LIN {X 0,Y 524.24,Z 195.314,A -85,B 0,C 180,E1 -4882.904,E2 -4882.904} C_VEL
LIN {X 0,Y 525.954,Z 203.789,A -85,B 0,C 180,E1 -4883.085,E2 -4883.085} C_VEL
LIN {X 0,Y 525.499,Z 302.73,A -85,B 0,C 180,E1 -4884.494,E2 -4884.494} C_VEL
LIN {X 0,Y 525.358,Z 316.211,A -85,B 0,C 180,E1 -4884.854,E2 -4884.854} C_VEL
LIN {X 0,Y 525.146,Z 328.864,A -85,B 0,C 180,E1 -4885.357,E2 -4885.357} C_VEL
LIN {X 0,Y 524.878,Z 340.909,A -85,B 0,C 180,E1 -4886.009,E2 -4886.009} C_VEL
LIN {X 0,Y 524.614,Z 351.923,A -85,B 0,C 180,E1 -4886.773,E2 -4886.773} C_VEL
LIN {X 0,Y 524.367,Z 361.654,A -85,B 0,C 180,E1 -4887.611,E2 -4887.611} C_VEL
LIN {X 0,Y 524.142,Z 371.309,A -85,B 0,C 180,E1 -4888.643,E2 -4888.643} C_VEL
LIN {X 0,Y 523.923,Z 379.749,A -85,B 0,C 180,E1 -4889.757,E2 -4889.757} C_VEL
LIN {X 0,Y 523.73,Z 386.278,A -85,B 0,C 180,E1 -4890.815,E2 -4890.815} C_VEL
LIN {X 0,Y 523.699,Z 387.83,A -85,B 0,C 180,E1 -4891.105,E2 -4891.105} C_VEL
LIN {X 0,Y 522.987,Z 390.737,A -85,B 0,C 180,E1 -4891.663,E2 -4891.663} C_VEL
LIN {X 0,Y 520.036,Z 395.032,A -85,B 0,C 180,E1 -4892.59,E2 -4892.59} C_VEL
LIN {X 0,Y 517.078,Z 398.654,A -85,B 0,C 180,E1 -4893.561,E2 -4893.561} C_VEL
LIN {X 0,Y 516.367,Z 400.435,A -85,B 0,C 180,E1 -4894.182,E2 -4894.182} C_VEL
LIN {X 0,Y 516.321,Z 402.767,A -85,B 0,C 180,E1 -4895.244,E2 -4895.244} C_VEL
LIN {X 0,Y 516.258,Z 404.817,A -85,B 0,C 180,E1 -4896.797,E2 -4896.797} C_VEL
LIN {X 0,Y 516.242,Z 405.275,A -85,B 0,C 180,E1 -4897.852,E2 -4897.852} C_VEL
LIN {X 0,Y 516.25,Z 404.907,A -85,B 0,C 180,E1 -4899.107,E2 -4899.107} C_VEL
LIN {X 0,Y 516.299,Z 403.557,A -85,B 0,C 180,E1 -4900.334,E2 -4900.334} C_VEL
LIN {X 0,Y 516.377,Z 400.571,A -85,B 0,C 180,E1 -4901.828,E2 -4901.828} C_VEL
LIN {X 0,Y 516.471,Z 397.517,A -85,B 0,C 180,E1 -4902.874,E2 -4902.874} C_VEL
LIN {X 0,Y 516.547,Z 392.428,A -85,B 0,C 180,E1 -4904.2,E2 -4904.2} C_VEL
LIN {X 0,Y 516.706,Z 385.586,A -85,B 0,C 180,E1 -4905.556,E2 -4905.556} C_VEL
LIN {X 0,Y 516.897,Z 378.682,A -85,B 0,C 180,E1 -4906.647,E2 -4906.647} C_VEL
LIN {X 0,Y 517.166,Z 370.161,A -85,B 0,C 180,E1 -4907.745,E2 -4907.745} C_VEL
LIN {X 0,Y 517.452,Z 359.972,A -85,B 0,C 180,E1 -4908.798,E2 -4908.798} C_VEL
LIN {X 0,Y 517.679,Z 349.531,A -85,B 0,C 180,E1 -4909.669,E2 -4909.669} C_VEL
LIN {X 0,Y 517.992,Z 338.867,A -85,B 0,C 180,E1 -4910.381,E2 -4910.381} C_VEL
LIN {X 0,Y 518.301,Z 327.456,A -85,B 0,C 180,E1 -4910.974,E2 -4910.974} C_VEL
LIN {X 0,Y 518.454,Z 313.875,A -85,B 0,C 180,E1 -4911.494,E2 -4911.494} C_VEL
LIN {X 0,Y 518.631,Z 301.35,A -85,B 0,C 180,E1 -4911.81,E2 -4911.81} C_VEL
LIN {X 0,Y 519.072,Z 204.764,A -85,B 0,C 180,E1 -4913.193,E2 -4913.193} C_VEL
LIN {X 0,Y 517.223,Z 195.581,A -85,B 0,C 180,E1 -4913.39,E2 -4913.39} C_VEL
LIN {X 0,Y 516.967,Z 190.248,A -85,B 0,C 180,E1 -4914.482,E2 -4914.482} C_VEL
LIN {X 0,Y 516.894,Z 190.102,A -85,B 0,C 180,E1 -4917.457,E2 -4917.457} C_VEL
LIN {X 0,Y 516.921,Z 190.092,A -85,B 0,C 180,E1 -4920.696,E2 -4920.696} C_VEL
LIN {X 0,Y 516.897,Z 190.094,A -85,B 0,C 180,E1 -4923.815,E2 -4923.815} C_VEL
LIN {X 0,Y 516.858,Z 190.103,A -85,B 0,C 180,E1 -4926.776,E2 -4926.776} C_VEL
LIN {X 0,Y 516.938,Z 190.088,A -85,B 0,C 180,E1 -4929.733,E2 -4929.733} C_VEL
LIN {X 0,Y 516.896,Z 190.097,A -85,B 0,C 180,E1 -4932.595,E2 -4932.595} C_VEL
LIN {X 0,Y 516.941,Z 190.094,A -85,B 0,C 180,E1 -4935.03,E2 -4935.03} C_VEL
LIN {X 0,Y 516.968,Z 190.086,A -85,B 0,C 180,E1 -4938.234,E2 -4938.234} C_VEL
LIN {X 0,Y 516.956,Z 190.086,A -85,B 0,C 180,E1 -4941.4,E2 -4941.4} C_VEL
LIN {X 0,Y 517.025,Z 190.085,A -85,B 0,C 180,E1 -4944.54,E2 -4944.54} C_VEL
LIN {X 0,Y 517.082,Z 190.07,A -85,B 0,C 180,E1 -4947.663,E2 -4947.663} C_VEL
LIN {X 0,Y 517.092,Z 190.073,A -85,B 0,C 180,E1 -4950.779,E2 -4950.779} C_VEL
LIN {X 0,Y 516.975,Z 190.084,A -85,B 0,C 180,E1 -4953.117,E2 -4953.117} C_VEL
LIN {X 0,Y 516.991,Z 190.089,A -85,B 0,C 180,E1 -4956.244,E2 -4956.244} C_VEL
LIN {X 0,Y 516.943,Z 190.087,A -85,B 0,C 180,E1 -4959.39,E2 -4959.39} C_VEL
LIN {X 0,Y 516.954,Z 190.089,A -85,B 0,C 180,E1 -4961.807,E2 -4961.807} C_VEL
LIN {X 0,Y 516.941,Z 190.087,A -85,B 0,C 180,E1 -4965.144,E2 -4965.144} C_VEL
LIN {X 0,Y 516.914,Z 190.098,A -85,B 0,C 180,E1 -4968.223,E2 -4968.223} C_VEL
LIN {X 0,Y 516.907,Z 190.093,A -85,B 0,C 180,E1 -4970.702,E2 -4970.702} C_VEL
LIN {X 0,Y 516.887,Z 190.101,A -85,B 0,C 180,E1 -4974.073,E2 -4974.073} C_VEL
LIN {X 0,Y 516.89,Z 190.094,A -85,B 0,C 180,E1 -4976.66,E2 -4976.66} C_VEL
LIN {X 0,Y 516.909,Z 190.096,A -85,B 0,C 180,E1 -4979.523,E2 -4979.523} C_VEL
LIN {X 0,Y 516.898,Z 190.093,A -85,B 0,C 180,E1 -4982.543,E2 -4982.543} C_VEL
LIN {X 0,Y 516.866,Z 190.101,A -85,B 0,C 180,E1 -4985.329,E2 -4985.329} C_VEL
LIN {X 0,Y 516.88,Z 190.099,A -85,B 0,C 180,E1 -4987.943,E2 -4987.943} C_VEL
LIN {X 0,Y 516.866,Z 190.097,A -85,B 0,C 180,E1 -4990.744,E2 -4990.744} C_VEL
LIN {X 0,Y 516.861,Z 190.099,A -85,B 0,C 180,E1 -4992.834,E2 -4992.834} C_VEL
LIN {X 0,Y 516.898,Z 190.096,A -85,B 0,C 180,E1 -4995.007,E2 -4995.007} C_VEL
LIN {X 0,Y 516.904,Z 190.092,A -85,B 0,C 180,E1 -4998.4,E2 -4998.4} C_VEL
LIN {X 0,Y 516.879,Z 190.105,A -85,B 0,C 180,E1 -5001.284,E2 -5001.284} C_VEL
LIN {X 0,Y 516.87,Z 190.096,A -85,B 0,C 180,E1 -5004.22,E2 -5004.22} C_VEL
LIN {X 0,Y 516.883,Z 190.102,A -85,B 0,C 180,E1 -5007.052,E2 -5007.052} C_VEL
LIN {X 0,Y 516.869,Z 190.097,A -85,B 0,C 180,E1 -5009.795,E2 -5009.795} C_VEL
LIN {X 0,Y 516.885,Z 190.096,A -85,B 0,C 180,E1 -5012.465,E2 -5012.465} C_VEL
LIN {X 0,Y 516.853,Z 190.106,A -85,B 0,C 180,E1 -5015.069,E2 -5015.069} C_VEL
LIN {X 0,Y 516.872,Z 190.097,A -85,B 0,C 180,E1 -5017.622,E2 -5017.622} C_VEL
LIN {X 0,Y 516.932,Z 190.089,A -85,B 0,C 180,E1 -5020.13,E2 -5020.13} C_VEL
LIN {X 0,Y 516.896,Z 190.099,A -85,B 0,C 180,E1 -5022.595,E2 -5022.595} C_VEL
LIN {X 0,Y 516.935,Z 190.093,A -85,B 0,C 180,E1 -5025.03,E2 -5025.03} C_VEL
LIN {X 0,Y 516.97,Z 190.087,A -85,B 0,C 180,E1 -5028.234,E2 -5028.234} C_VEL
LIN {X 0,Y 516.956,Z 190.086,A -85,B 0,C 180,E1 -5031.399,E2 -5031.399} C_VEL
LIN {X 0,Y 517.014,Z 190.087,A -85,B 0,C 180,E1 -5034.54,E2 -5034.54} C_VEL
LIN {X 0,Y 517.082,Z 190.07,A -85,B 0,C 180,E1 -5037.663,E2 -5037.663} C_VEL
LIN {X 0,Y 517.069,Z 190.075,A -85,B 0,C 180,E1 -5040.779,E2 -5040.779} C_VEL
LIN {X 0,Y 516.949,Z 190.087,A -85,B 0,C 180,E1 -5043.117,E2 -5043.117} C_VEL
LIN {X 0,Y 516.975,Z 190.092,A -85,B 0,C 180,E1 -5046.244,E2 -5046.244} C_VEL
LIN {X 0,Y 516.939,Z 190.088,A -85,B 0,C 180,E1 -5049.39,E2 -5049.39} C_VEL
LIN {X 0,Y 516.956,Z 190.091,A -85,B 0,C 180,E1 -5051.807,E2 -5051.807} C_VEL
LIN {X 0,Y 516.943,Z 190.087,A -85,B 0,C 180,E1 -5055.144,E2 -5055.144} C_VEL
LIN {X 0,Y 516.879,Z 190.1,A -85,B 0,C 180,E1 -5058.224,E2 -5058.224} C_VEL
LIN {X 0,Y 516.903,Z 190.093,A -85,B 0,C 180,E1 -5060.702,E2 -5060.702} C_VEL
LIN {X 0,Y 516.859,Z 190.099,A -85,B 0,C 180,E1 -5063.224,E2 -5063.224} C_VEL
LIN {X 0,Y 516.884,Z 190.097,A -85,B 0,C 180,E1 -5066.182,E2 -5066.182} C_VEL
LIN {X 0,Y 516.906,Z 190.096,A -85,B 0,C 180,E1 -5069.306,E2 -5069.306} C_VEL
LIN {X 0,Y 516.896,Z 190.093,A -85,B 0,C 180,E1 -5072.543,E2 -5072.543} C_VEL
LIN {X 0,Y 516.863,Z 190.103,A -85,B 0,C 180,E1 -5075.328,E2 -5075.328} C_VEL
LIN {X 0,Y 516.88,Z 190.098,A -85,B 0,C 180,E1 -5077.942,E2 -5077.942} C_VEL
LIN {X 0,Y 516.855,Z 190.099,A -85,B 0,C 180,E1 -5080.745,E2 -5080.745} C_VEL
LIN {X 0,Y 516.883,Z 190.096,A -85,B 0,C 180,E1 -5083.903,E2 -5083.903} C_VEL
LIN {X 0,Y 516.882,Z 190.095,A -85,B 0,C 180,E1 -5086.107,E2 -5086.107} C_VEL
LIN {X 0,Y 516.855,Z 190.106,A -85,B 0,C 180,E1 -5089.255,E2 -5089.255} C_VEL
LIN {X 0,Y 516.862,Z 190.098,A -85,B 0,C 180,E1 -5092.274,E2 -5092.274} C_VEL
LIN {X 0,Y 516.875,Z 190.104,A -85,B 0,C 180,E1 -5095.174,E2 -5095.174} C_VEL
LIN {X 0,Y 516.87,Z 190.098,A -85,B 0,C 180,E1 -5097.974,E2 -5097.974} C_VEL
LIN {X 0,Y 516.905,Z 190.099,A -85,B 0,C 180,E1 -5100.694,E2 -5100.694} C_VEL
LIN {X 0,Y 516.901,Z 190.178,A -85,B 0,C 180,E1 -5103.633,E2 -5103.633} C_VEL
LIN {X 0,Y 518.785,Z 200.2,A -85,B 0,C 180,E1 -5105.183,E2 -5105.183} C_VEL
LIN {X 0,Y 518.36,Z 217.704,A -85,B 0,C 180,E1 -5107.689,E2 -5107.689} C_VEL
LIN {X 0,Y 517.906,Z 238.22,A -85,B 0,C 180,E1 -5110.581,E2 -5110.581} C_VEL
LIN {X 0,Y 517.415,Z 260.123,A -85,B 0,C 180,E1 -5113.629,E2 -5113.629} C_VEL
LIN {X 0,Y 517.252,Z 267.307,A -85,B 0,C 180,E1 -5114.623,E2 -5114.623} C_VEL
LIN {X 0,Y 519.019,Z 280.709,A -85,B 0,C 180,E1 -5114.873,E2 -5114.873} C_VEL
LIN {X 0,Y 518.492,Z 377.185,A -85,B 0,C 180,E1 -5116.253,E2 -5116.253} C_VEL
LIN {X 0,Y 518.229,Z 390.964,A -85,B 0,C 180,E1 -5116.621,E2 -5116.621} C_VEL
LIN {X 0,Y 517.971,Z 403.375,A -85,B 0,C 180,E1 -5117.113,E2 -5117.113} C_VEL
LIN {X 0,Y 517.622,Z 415.512,A -85,B 0,C 180,E1 -5117.766,E2 -5117.766} C_VEL
LIN {X 0,Y 517.352,Z 426.757,A -85,B 0,C 180,E1 -5118.54,E2 -5118.54} C_VEL
LIN {X 0,Y 517.081,Z 437.113,A -85,B 0,C 180,E1 -5119.427,E2 -5119.427} C_VEL
LIN {X 0,Y 516.812,Z 446.415,A -85,B 0,C 180,E1 -5120.41,E2 -5120.41} C_VEL
LIN {X 0,Y 516.628,Z 455.472,A -85,B 0,C 180,E1 -5121.591,E2 -5121.591} C_VEL
LIN {X 0,Y 516.503,Z 462.768,A -85,B 0,C 180,E1 -5122.769,E2 -5122.769} C_VEL
LIN {X 0,Y 516.381,Z 467.688,A -85,B 0,C 180,E1 -5123.749,E2 -5123.749} C_VEL
LIN {X 0,Y 516.312,Z 472.473,A -85,B 0,C 180,E1 -5124.924,E2 -5124.924} C_VEL
LIN {X 0,Y 516.372,Z 476.135,A -85,B 0,C 180,E1 -5126.098,E2 -5126.098} C_VEL
LIN {X 0,Y 516.346,Z 478.019,A -85,B 0,C 180,E1 -5126.879,E2 -5126.879} C_VEL
LIN {X 0,Y 516.264,Z 479.427,A -85,B 0,C 180,E1 -5127.659,E2 -5127.659} C_VEL
LIN {X 0,Y 516.199,Z 481.039,A -85,B 0,C 180,E1 -5129.22,E2 -5129.22} C_VEL
LIN {X 0,Y 516.203,Z 481.252,A -85,B 0,C 180,E1 -5130,E2 -5130} C_VEL
LIN {X 0,Y 516.2,Z 481.027,A -85,B 0,C 180,E1 -5130.78,E2 -5130.78} C_VEL
LIN {X 0,Y 516.264,Z 479.391,A -85,B 0,C 180,E1 -5132.34,E2 -5132.34} C_VEL
LIN {X 0,Y 516.362,Z 477.97,A -85,B 0,C 180,E1 -5133.121,E2 -5133.121} C_VEL
LIN {X 0,Y 516.344,Z 474.975,A -85,B 0,C 180,E1 -5134.293,E2 -5134.293} C_VEL
LIN {X 0,Y 516.389,Z 470.928,A -85,B 0,C 180,E1 -5135.467,E2 -5135.467} C_VEL
LIN {X 0,Y 516.418,Z 465.656,A -85,B 0,C 180,E1 -5136.655,E2 -5136.655} C_VEL
LIN {X 0,Y 516.538,Z 459.159,A -85,B 0,C 180,E1 -5137.82,E2 -5137.82} C_VEL
LIN {X 0,Y 516.713,Z 450.992,A -85,B 0,C 180,E1 -5138.999,E2 -5138.999} C_VEL
LIN {X 0,Y 516.903,Z 442.664,A -85,B 0,C 180,E1 -5139.983,E2 -5139.983} C_VEL
LIN {X 0,Y 517.199,Z 432.511,A -85,B 0,C 180,E1 -5140.967,E2 -5140.967} C_VEL
LIN {X 0,Y 517.446,Z 421.234,A -85,B 0,C 180,E1 -5141.84,E2 -5141.84} C_VEL
LIN {X 0,Y 517.789,Z 409.771,A -85,B 0,C 180,E1 -5142.543,E2 -5142.543} C_VEL
LIN {X 0,Y 518.077,Z 397.232,A -85,B 0,C 180,E1 -5143.133,E2 -5143.133} C_VEL
LIN {X 0,Y 518.353,Z 383.87,A -85,B 0,C 180,E1 -5143.575,E2 -5143.575} C_VEL
LIN {X 0,Y 518.583,Z 370.916,A -85,B 0,C 180,E1 -5143.844,E2 -5143.844} C_VEL
LIN {X 0,Y 518.922,Z 279.596,A -85,B 0,C 180,E1 -5145.138,E2 -5145.138} C_VEL
LIN {X 0,Y 517.22,Z 266.453,A -85,B 0,C 180,E1 -5145.397,E2 -5145.397} C_VEL
LIN {X 0,Y 517.663,Z 242.885,A -85,B 0,C 180,E1 -5148.605,E2 -5148.605} C_VEL
LIN {X 0,Y 517.991,Z 221.824,A -85,B 0,C 180,E1 -5151.489,E2 -5151.489} C_VEL
LIN {X 0,Y 518.421,Z 200.841,A -85,B 0,C 180,E1 -5154.386,E2 -5154.386} C_VEL
LIN {X 0,Y 518.054,Z 195.968,A -85,B 0,C 180,E1 -5155.084,E2 -5155.084} C_VEL
LIN {X 0,Y 516.884,Z 190.1,A -85,B 0,C 180,E1 -5155.985,E2 -5155.985} C_VEL
LIN {X 0,Y 516.849,Z 190.104,A -85,B 0,C 180,E1 -5158.419,E2 -5158.419} C_VEL
LIN {X 0,Y 516.88,Z 190.104,A -85,B 0,C 180,E1 -5161.11,E2 -5161.11} C_VEL
LIN {X 0,Y 516.886,Z 190.096,A -85,B 0,C 180,E1 -5163.962,E2 -5163.962} C_VEL
LIN {X 0,Y 516.854,Z 190.107,A -85,B 0,C 180,E1 -5166.748,E2 -5166.748} C_VEL
LIN {X 0,Y 516.858,Z 190.099,A -85,B 0,C 180,E1 -5169.723,E2 -5169.723} C_VEL
LIN {X 0,Y 516.901,Z 190.093,A -85,B 0,C 180,E1 -5171.776,E2 -5171.776} C_VEL
LIN {X 0,Y 516.896,Z 190.097,A -85,B 0,C 180,E1 -5175.007,E2 -5175.007} C_VEL
LIN {X 0,Y 516.903,Z 190.099,A -85,B 0,C 180,E1 -5178.4,E2 -5178.4} C_VEL
LIN {X 0,Y 516.877,Z 190.097,A -85,B 0,C 180,E1 -5181.284,E2 -5181.284} C_VEL
LIN {X 0,Y 516.868,Z 190.105,A -85,B 0,C 180,E1 -5184.219,E2 -5184.219} C_VEL
LIN {X 0,Y 516.895,Z 190.094,A -85,B 0,C 180,E1 -5187.053,E2 -5187.053} C_VEL
LIN {X 0,Y 516.885,Z 190.099,A -85,B 0,C 180,E1 -5189.796,E2 -5189.796} C_VEL
LIN {X 0,Y 516.899,Z 190.096,A -85,B 0,C 180,E1 -5192.466,E2 -5192.466} C_VEL
LIN {X 0,Y 516.851,Z 190.1,A -85,B 0,C 180,E1 -5195.069,E2 -5195.069} C_VEL
LIN {X 0,Y 516.869,Z 190.1,A -85,B 0,C 180,E1 -5197.621,E2 -5197.621} C_VEL
LIN {X 0,Y 516.929,Z 190.096,A -85,B 0,C 180,E1 -5200.13,E2 -5200.13} C_VEL
LIN {X 0,Y 516.894,Z 190.093,A -85,B 0,C 180,E1 -5202.595,E2 -5202.595} C_VEL
LIN {X 0,Y 516.936,Z 190.089,A -85,B 0,C 180,E1 -5205.03,E2 -5205.03} C_VEL
LIN {X 0,Y 516.966,Z 190.086,A -85,B 0,C 180,E1 -5208.234,E2 -5208.234} C_VEL
LIN {X 0,Y 516.965,Z 190.09,A -85,B 0,C 180,E1 -5211.4,E2 -5211.4} C_VEL
LIN {X 0,Y 517.003,Z 190.086,A -85,B 0,C 180,E1 -5213.757,E2 -5213.757} C_VEL
LIN {X 0,Y 517.009,Z 190.081,A -85,B 0,C 180,E1 -5216.883,E2 -5216.883} C_VEL
LIN {X 0,Y 517.093,Z 190.075,A -85,B 0,C 180,E1 -5219.221,E2 -5219.221} C_VEL
LIN {X 0,Y 517.084,Z 190.071,A -85,B 0,C 180,E1 -5222.337,E2 -5222.337} C_VEL
LIN {X 0,Y 517.027,Z 190.083,A -85,B 0,C 180,E1 -5225.46,E2 -5225.46} C_VEL
LIN {X 0,Y 516.956,Z 190.089,A -85,B 0,C 180,E1 -5228.6,E2 -5228.6} C_VEL
LIN {X 0,Y 516.952,Z 190.09,A -85,B 0,C 180,E1 -5231.807,E2 -5231.807} C_VEL
LIN {X 0,Y 516.945,Z 190.096,A -85,B 0,C 180,E1 -5235.146,E2 -5235.146} C_VEL
LIN {X 0,Y 516.916,Z 190.095,A -85,B 0,C 180,E1 -5238.223,E2 -5238.223} C_VEL
LIN {X 0,Y 516.919,Z 190.099,A -85,B 0,C 180,E1 -5240.701,E2 -5240.701} C_VEL
LIN {X 0,Y 516.949,Z 190.192,A -85,B 0,C 180,E1 -5241.666,E2 -5241.666} C_VEL
LIN {X 0,Y 517.31,Z 195.958,A -85,B 0,C 180,E1 -5242.705,E2 -5242.705} C_VEL
LIN {X 0,Y 519.135,Z 204.977,A -85,B 0,C 180,E1 -5242.894,E2 -5242.894} C_VEL
LIN {X 0,Y 518.632,Z 302.232,A -85,B 0,C 180,E1 -5244.295,E2 -5244.295} C_VEL
LIN {X 0,Y 518.454,Z 315.813,A -85,B 0,C 180,E1 -5244.651,E2 -5244.651} C_VEL
LIN {X 0,Y 518.259,Z 327.987,A -85,B 0,C 180,E1 -5245.127,E2 -5245.127} C_VEL
LIN {X 0,Y 518.039,Z 339.471,A -85,B 0,C 180,E1 -5245.73,E2 -5245.73} C_VEL
LIN {X 0,Y 517.687,Z 351.282,A -85,B 0,C 180,E1 -5246.535,E2 -5246.535} C_VEL
LIN {X 0,Y 517.426,Z 361.324,A -85,B 0,C 180,E1 -5247.394,E2 -5247.394} C_VEL
LIN {X 0,Y 517.173,Z 370.859,A -85,B 0,C 180,E1 -5248.4,E2 -5248.4} C_VEL
LIN {X 0,Y 516.912,Z 379.436,A -85,B 0,C 180,E1 -5249.524,E2 -5249.524} C_VEL
LIN {X 0,Y 516.702,Z 387.362,A -85,B 0,C 180,E1 -5250.819,E2 -5250.819} C_VEL
LIN {X 0,Y 516.564,Z 393.243,A -85,B 0,C 180,E1 -5252.046,E2 -5252.046} C_VEL
LIN {X 0,Y 516.449,Z 398.293,A -85,B 0,C 180,E1 -5253.427,E2 -5253.427} C_VEL
LIN {X 0,Y 516.367,Z 400.435,A -85,B 0,C 180,E1 -5254.182,E2 -5254.182} C_VEL
LIN {X 0,Y 515.672,Z 402.003,A -85,B 0,C 180,E1 -5254.81,E2 -5254.81} C_VEL
LIN {X 0,Y 512.779,Z 404.107,A -85,B 0,C 180,E1 -5255.841,E2 -5255.841} C_VEL
LIN {X 0,Y 510.337,Z 405.224,A -85,B 0,C 180,E1 -5256.682,E2 -5256.682} C_VEL
LIN {X 0,Y 509.268,Z 405.667,A -85,B 0,C 180,E1 -5257.336,E2 -5257.336} C_VEL
LIN {X 0,Y 509.17,Z 405.728,A -85,B 0,C 180,E1 -5257.558,E2 -5257.558} C_VEL
LIN {X 0,Y 509.145,Z 405.758,A -85,B 0,C 180,E1 -5258.401,E2 -5258.401} C_VEL
LIN {X 0,Y 509.177,Z 405.206,A -85,B 0,C 180,E1 -5259.414,E2 -5259.414} C_VEL
LIN {X 0,Y 509.219,Z 403.697,A -85,B 0,C 180,E1 -5260.617,E2 -5260.617} C_VEL
LIN {X 0,Y 509.324,Z 401.204,A -85,B 0,C 180,E1 -5261.83,E2 -5261.83} C_VEL
LIN {X 0,Y 509.423,Z 396.845,A -85,B 0,C 180,E1 -5263.282,E2 -5263.282} C_VEL
LIN {X 0,Y 509.574,Z 391.035,A -85,B 0,C 180,E1 -5264.699,E2 -5264.699} C_VEL
LIN {X 0,Y 509.696,Z 385.232,A -85,B 0,C 180,E1 -5265.808,E2 -5265.808} C_VEL
LIN {X 0,Y 509.927,Z 378.047,A -85,B 0,C 180,E1 -5266.925,E2 -5266.925} C_VEL
LIN {X 0,Y 510.227,Z 369.028,A -85,B 0,C 180,E1 -5268.057,E2 -5268.057} C_VEL
LIN {X 0,Y 510.573,Z 358.475,A -85,B 0,C 180,E1 -5269.125,E2 -5269.125} C_VEL
LIN {X 0,Y 510.836,Z 347.824,A -85,B 0,C 180,E1 -5269.983,E2 -5269.983} C_VEL
LIN {X 0,Y 511.179,Z 335.381,A -85,B 0,C 180,E1 -5270.77,E2 -5270.77} C_VEL
LIN {X 0,Y 511.491,Z 324.034,A -85,B 0,C 180,E1 -5271.318,E2 -5271.318} C_VEL
LIN {X 0,Y 511.65,Z 311.026,A -85,B 0,C 180,E1 -5271.77,E2 -5271.77} C_VEL
LIN {X 0,Y 511.772,Z 298.423,A -85,B 0,C 180,E1 -5272.05,E2 -5272.05} C_VEL
LIN {X 0,Y 512.193,Z 205.45,A -85,B 0,C 180,E1 -5273.398,E2 -5273.398} C_VEL
LIN {X 0,Y 510.256,Z 195.913,A -85,B 0,C 180,E1 -5273.613,E2 -5273.613} C_VEL
LIN {X 0,Y 509.883,Z 190.979,A -85,B 0,C 180,E1 -5274.626,E2 -5274.626} C_VEL
LIN {X 0,Y 509.86,Z 190.978,A -85,B 0,C 180,E1 -5277.481,E2 -5277.481} C_VEL
LIN {X 0,Y 509.859,Z 190.97,A -85,B 0,C 180,E1 -5280.274,E2 -5280.274} C_VEL
LIN {X 0,Y 509.866,Z 190.975,A -85,B 0,C 180,E1 -5282.943,E2 -5282.943} C_VEL
LIN {X 0,Y 509.838,Z 190.975,A -85,B 0,C 180,E1 -5285.573,E2 -5285.573} C_VEL
LIN {X 0,Y 509.822,Z 190.974,A -85,B 0,C 180,E1 -5288.149,E2 -5288.149} C_VEL
LIN {X 0,Y 509.858,Z 190.975,A -85,B 0,C 180,E1 -5290.682,E2 -5290.682} C_VEL
LIN {X 0,Y 509.865,Z 190.974,A -85,B 0,C 180,E1 -5293.174,E2 -5293.174} C_VEL
LIN {X 0,Y 509.858,Z 190.97,A -85,B 0,C 180,E1 -5295.634,E2 -5295.634} C_VEL
LIN {X 0,Y 509.914,Z 190.97,A -85,B 0,C 180,E1 -5298.875,E2 -5298.875} C_VEL
LIN {X 0,Y 509.922,Z 190.963,A -85,B 0,C 180,E1 -5302.078,E2 -5302.078} C_VEL
LIN {X 0,Y 509.976,Z 190.961,A -85,B 0,C 180,E1 -5304.464,E2 -5304.464} C_VEL
LIN {X 0,Y 510.052,Z 190.946,A -85,B 0,C 180,E1 -5307.631,E2 -5307.631} C_VEL
LIN {X 0,Y 510.063,Z 190.949,A -85,B 0,C 180,E1 -5310.79,E2 -5310.79} C_VEL
LIN {X 0,Y 509.918,Z 190.963,A -85,B 0,C 180,E1 -5313.161,E2 -5313.161} C_VEL
LIN {X 0,Y 509.939,Z 190.969,A -85,B 0,C 180,E1 -5316.33,E2 -5316.33} C_VEL
LIN {X 0,Y 509.911,Z 190.966,A -85,B 0,C 180,E1 -5318.721,E2 -5318.721} C_VEL
LIN {X 0,Y 509.907,Z 190.968,A -85,B 0,C 180,E1 -5321.932,E2 -5321.932} C_VEL
LIN {X 0,Y 509.897,Z 190.965,A -85,B 0,C 180,E1 -5325.242,E2 -5325.242} C_VEL
LIN {X 0,Y 509.858,Z 190.973,A -85,B 0,C 180,E1 -5328.484,E2 -5328.484} C_VEL
LIN {X 0,Y 509.848,Z 190.971,A -85,B 0,C 180,E1 -5331.002,E2 -5331.002} C_VEL
LIN {X 0,Y 509.821,Z 190.978,A -85,B 0,C 180,E1 -5333.564,E2 -5333.564} C_VEL
LIN {X 0,Y 509.873,Z 190.97,A -85,B 0,C 180,E1 -5336.369,E2 -5336.369} C_VEL
LIN {X 0,Y 509.86,Z 190.978,A -85,B 0,C 180,E1 -5339.726,E2 -5339.726} C_VEL
LIN {X 0,Y 509.875,Z 190.968,A -85,B 0,C 180,E1 -5342.774,E2 -5342.774} C_VEL
LIN {X 0,Y 509.825,Z 190.982,A -85,B 0,C 180,E1 -5345.578,E2 -5345.578} C_VEL
LIN {X 0,Y 509.85,Z 190.971,A -85,B 0,C 180,E1 -5348.338,E2 -5348.338} C_VEL
LIN {X 0,Y 509.847,Z 190.979,A -85,B 0,C 180,E1 -5351.427,E2 -5351.427} C_VEL
LIN {X 0,Y 509.841,Z 190.972,A -85,B 0,C 180,E1 -5354.67,E2 -5354.67} C_VEL
LIN {X 0,Y 509.847,Z 190.972,A -85,B 0,C 180,E1 -5358.105,E2 -5358.105} C_VEL
LIN {X 0,Y 509.835,Z 190.974,A -85,B 0,C 180,E1 -5360.646,E2 -5360.646} C_VEL
LIN {X 0,Y 509.812,Z 190.979,A -85,B 0,C 180,E1 -5363.646,E2 -5363.646} C_VEL
LIN {X 0,Y 509.844,Z 190.973,A -85,B 0,C 180,E1 -5366.538,E2 -5366.538} C_VEL
LIN {X 0,Y 509.836,Z 190.978,A -85,B 0,C 180,E1 -5369.334,E2 -5369.334} C_VEL
LIN {X 0,Y 509.84,Z 190.972,A -85,B 0,C 180,E1 -5372.051,E2 -5372.051} C_VEL
LIN {X 0,Y 509.811,Z 190.981,A -85,B 0,C 180,E1 -5374.7,E2 -5374.7} C_VEL
LIN {X 0,Y 509.828,Z 190.975,A -85,B 0,C 180,E1 -5377.459,E2 -5377.459} C_VEL
LIN {X 0,Y 509.918,Z 190.962,A -85,B 0,C 180,E1 -5379.845,E2 -5379.845} C_VEL
LIN {X 0,Y 509.861,Z 190.973,A -85,B 0,C 180,E1 -5383.174,E2 -5383.174} C_VEL
LIN {X 0,Y 509.85,Z 190.971,A -85,B 0,C 180,E1 -5385.634,E2 -5385.634} C_VEL
LIN {X 0,Y 509.915,Z 190.968,A -85,B 0,C 180,E1 -5388.875,E2 -5388.875} C_VEL
LIN {X 0,Y 509.911,Z 190.966,A -85,B 0,C 180,E1 -5392.078,E2 -5392.078} C_VEL
LIN {X 0,Y 509.965,Z 190.965,A -85,B 0,C 180,E1 -5394.464,E2 -5394.464} C_VEL
LIN {X 0,Y 510.052,Z 190.946,A -85,B 0,C 180,E1 -5397.631,E2 -5397.631} C_VEL
LIN {X 0,Y 510.021,Z 190.952,A -85,B 0,C 180,E1 -5400.79,E2 -5400.79} C_VEL
LIN {X 0,Y 510.047,Z 190.954,A -85,B 0,C 180,E1 -5402.369,E2 -5402.369} C_VEL
LIN {X 0,Y 509.944,Z 190.96,A -85,B 0,C 180,E1 -5405.536,E2 -5405.536} C_VEL
LIN {X 0,Y 509.888,Z 190.968,A -85,B 0,C 180,E1 -5408.721,E2 -5408.721} C_VEL
LIN {X 0,Y 509.908,Z 190.97,A -85,B 0,C 180,E1 -5411.932,E2 -5411.932} C_VEL
LIN {X 0,Y 509.898,Z 190.965,A -85,B 0,C 180,E1 -5415.242,E2 -5415.242} C_VEL
LIN {X 0,Y 509.838,Z 190.974,A -85,B 0,C 180,E1 -5418.485,E2 -5418.485} C_VEL
LIN {X 0,Y 509.845,Z 190.972,A -85,B 0,C 180,E1 -5421.002,E2 -5421.002} C_VEL
LIN {X 0,Y 509.821,Z 190.98,A -85,B 0,C 180,E1 -5423.564,E2 -5423.564} C_VEL
LIN {X 0,Y 509.821,Z 190.976,A -85,B 0,C 180,E1 -5426.357,E2 -5426.357} C_VEL
LIN {X 0,Y 509.839,Z 190.972,A -85,B 0,C 180,E1 -5428.847,E2 -5428.847} C_VEL
LIN {X 0,Y 509.821,Z 190.983,A -85,B 0,C 180,E1 -5431.59,E2 -5431.59} C_VEL
LIN {X 0,Y 509.837,Z 190.973,A -85,B 0,C 180,E1 -5434.415,E2 -5434.415} C_VEL
LIN {X 0,Y 509.81,Z 190.983,A -85,B 0,C 180,E1 -5437.342,E2 -5437.342} C_VEL
LIN {X 0,Y 509.817,Z 190.975,A -85,B 0,C 180,E1 -5440.385,E2 -5440.385} C_VEL
LIN {X 0,Y 509.808,Z 190.981,A -85,B 0,C 180,E1 -5443.573,E2 -5443.573} C_VEL
LIN {X 0,Y 509.808,Z 190.976,A -85,B 0,C 180,E1 -5446.426,E2 -5446.426} C_VEL
LIN {X 0,Y 509.816,Z 190.978,A -85,B 0,C 180,E1 -5449.615,E2 -5449.615} C_VEL
LIN {X 0,Y 509.81,Z 190.979,A -85,B 0,C 180,E1 -5452.658,E2 -5452.658} C_VEL
LIN {X 0,Y 509.841,Z 190.972,A -85,B 0,C 180,E1 -5455.8,E2 -5455.8} C_VEL
LIN {X 0,Y 509.841,Z 190.979,A -85,B 0,C 180,E1 -5458.722,E2 -5458.722} C_VEL
LIN {X 0,Y 509.839,Z 190.98,A -85,B 0,C 180,E1 -5461.153,E2 -5461.153} C_VEL
LIN {X 0,Y 509.869,Z 191.075,A -85,B 0,C 180,E1 -5463.447,E2 -5463.447} C_VEL
LIN {X 0,Y 511.9,Z 201.811,A -85,B 0,C 180,E1 -5465.131,E2 -5465.131} C_VEL
LIN {X 0,Y 511.391,Z 220.177,A -85,B 0,C 180,E1 -5467.794,E2 -5467.794} C_VEL
LIN {X 0,Y 510.856,Z 242.123,A -85,B 0,C 180,E1 -5470.929,E2 -5470.929} C_VEL
LIN {X 0,Y 510.282,Z 265.583,A -85,B 0,C 180,E1 -5474.233,E2 -5474.233} C_VEL
LIN {X 0,Y 510.241,Z 266.88,A -85,B 0,C 180,E1 -5474.411,E2 -5474.411} C_VEL
LIN {X 0,Y 512.17,Z 281.29,A -85,B 0,C 180,E1 -5474.681,E2 -5474.681} C_VEL
LIN {X 0,Y 511.604,Z 376.413,A -85,B 0,C 180,E1 -5476.064,E2 -5476.064} C_VEL
LIN {X 0,Y 511.292,Z 390.272,A -85,B 0,C 180,E1 -5476.436,E2 -5476.436} C_VEL
LIN {X 0,Y 511.015,Z 402.741,A -85,B 0,C 180,E1 -5476.934,E2 -5476.934} C_VEL
LIN {X 0,Y 510.684,Z 414.594,A -85,B 0,C 180,E1 -5477.577,E2 -5477.577} C_VEL
LIN {X 0,Y 510.354,Z 424.868,A -85,B 0,C 180,E1 -5478.28,E2 -5478.28} C_VEL
LIN {X 0,Y 510.133,Z 435.476,A -85,B 0,C 180,E1 -5479.181,E2 -5479.181} C_VEL
LIN {X 0,Y 509.81,Z 444.141,A -85,B 0,C 180,E1 -5480.077,E2 -5480.077} C_VEL
LIN {X 0,Y 509.627,Z 452.144,A -85,B 0,C 180,E1 -5481.075,E2 -5481.075} C_VEL
LIN {X 0,Y 509.428,Z 459.966,A -85,B 0,C 180,E1 -5482.269,E2 -5482.269} C_VEL
LIN {X 0,Y 509.309,Z 466.333,A -85,B 0,C 180,E1 -5483.483,E2 -5483.483} C_VEL
LIN {X 0,Y 509.244,Z 471.95,A -85,B 0,C 180,E1 -5484.853,E2 -5484.853} C_VEL
LIN {X 0,Y 509.3,Z 475.616,A -85,B 0,C 180,E1 -5486.043,E2 -5486.043} C_VEL
LIN {X 0,Y 509.258,Z 477.5,A -85,B 0,C 180,E1 -5486.835,E2 -5486.835} C_VEL
LIN {X 0,Y 509.195,Z 478.911,A -85,B 0,C 180,E1 -5487.627,E2 -5487.627} C_VEL
LIN {X 0,Y 509.117,Z 480.52,A -85,B 0,C 180,E1 -5489.209,E2 -5489.209} C_VEL
LIN {X 0,Y 509.123,Z 480.732,A -85,B 0,C 180,E1 -5490,E2 -5490} C_VEL
LIN {X 0,Y 509.118,Z 480.505,A -85,B 0,C 180,E1 -5490.791,E2 -5490.791} C_VEL
LIN {X 0,Y 509.196,Z 478.861,A -85,B 0,C 180,E1 -5492.373,E2 -5492.373} C_VEL
LIN {X 0,Y 509.273,Z 477.435,A -85,B 0,C 180,E1 -5493.164,E2 -5493.164} C_VEL
LIN {X 0,Y 509.252,Z 474.431,A -85,B 0,C 180,E1 -5494.353,E2 -5494.353} C_VEL
LIN {X 0,Y 509.3,Z 470.374,A -85,B 0,C 180,E1 -5495.543,E2 -5495.543} C_VEL
LIN {X 0,Y 509.368,Z 464.238,A -85,B 0,C 180,E1 -5496.914,E2 -5496.914} C_VEL
LIN {X 0,Y 509.489,Z 457.322,A -85,B 0,C 180,E1 -5498.128,E2 -5498.128} C_VEL
LIN {X 0,Y 509.689,Z 448.876,A -85,B 0,C 180,E1 -5499.324,E2 -5499.324} C_VEL
LIN {X 0,Y 509.92,Z 440.2,A -85,B 0,C 180,E1 -5500.321,E2 -5500.321} C_VEL
LIN {X 0,Y 510.248,Z 429.504,A -85,B 0,C 180,E1 -5501.319,E2 -5501.319} C_VEL
LIN {X 0,Y 510.523,Z 417.701,A -85,B 0,C 180,E1 -5502.202,E2 -5502.202} C_VEL
LIN {X 0,Y 510.848,Z 406.25,A -85,B 0,C 180,E1 -5502.867,E2 -5502.867} C_VEL
LIN {X 0,Y 511.196,Z 393.86,A -85,B 0,C 180,E1 -5503.415,E2 -5503.415} C_VEL
LIN {X 0,Y 511.48,Z 381.207,A -85,B 0,C 180,E1 -5503.812,E2 -5503.812} C_VEL
LIN {X 0,Y 511.686,Z 368.217,A -85,B 0,C 180,E1 -5504.06,E2 -5504.06} C_VEL
LIN {X 0,Y 512.013,Z 279.897,A -85,B 0,C 180,E1 -5505.333,E2 -5505.333} C_VEL
LIN {X 0,Y 510.173,Z 265.902,A -85,B 0,C 180,E1 -5505.609,E2 -5505.609} C_VEL
LIN {X 0,Y 510.703,Z 242.262,A -85,B 0,C 180,E1 -5508.868,E2 -5508.868} C_VEL
LIN {X 0,Y 511.046,Z 221.158,A -85,B 0,C 180,E1 -5511.796,E2 -5511.796} C_VEL
LIN {X 0,Y 511.474,Z 201.044,A -85,B 0,C 180,E1 -5514.62,E2 -5514.62} C_VEL
LIN {X 0,Y 510.721,Z 195.291,A -85,B 0,C 180,E1 -5515.469,E2 -5515.469} C_VEL
LIN {X 0,Y 509.868,Z 190.974,A -85,B 0,C 180,E1 -5516.146,E2 -5516.146} C_VEL
LIN {X 0,Y 509.837,Z 190.982,A -85,B 0,C 180,E1 -5518.847,E2 -5518.847} C_VEL
LIN {X 0,Y 509.812,Z 190.979,A -85,B 0,C 180,E1 -5521.591,E2 -5521.591} C_VEL
LIN {X 0,Y 509.838,Z 190.977,A -85,B 0,C 180,E1 -5524.414,E2 -5524.414} C_VEL
LIN {X 0,Y 509.808,Z 190.979,A -85,B 0,C 180,E1 -5527.341,E2 -5527.341} C_VEL
LIN {X 0,Y 509.818,Z 190.98,A -85,B 0,C 180,E1 -5530.384,E2 -5530.384} C_VEL
LIN {X 0,Y 509.801,Z 190.981,A -85,B 0,C 180,E1 -5533.059,E2 -5533.059} C_VEL
LIN {X 0,Y 509.822,Z 190.975,A -85,B 0,C 180,E1 -5535.793,E2 -5535.793} C_VEL
LIN {X 0,Y 509.845,Z 190.98,A -85,B 0,C 180,E1 -5538.573,E2 -5538.573} C_VEL
LIN {X 0,Y 509.849,Z 190.973,A -85,B 0,C 180,E1 -5541.787,E2 -5541.787} C_VEL
LIN {X 0,Y 509.828,Z 190.978,A -85,B 0,C 180,E1 -5544.622,E2 -5544.622} C_VEL
LIN {X 0,Y 509.861,Z 190.97,A -85,B 0,C 180,E1 -5547.481,E2 -5547.481} C_VEL
LIN {X 0,Y 509.858,Z 190.976,A -85,B 0,C 180,E1 -5550.274,E2 -5550.274} C_VEL
LIN {X 0,Y 509.859,Z 190.969,A -85,B 0,C 180,E1 -5552.943,E2 -5552.943} C_VEL
LIN {X 0,Y 509.838,Z 190.976,A -85,B 0,C 180,E1 -5555.572,E2 -5555.572} C_VEL
LIN {X 0,Y 509.822,Z 190.981,A -85,B 0,C 180,E1 -5558.148,E2 -5558.148} C_VEL
LIN {X 0,Y 509.856,Z 190.971,A -85,B 0,C 180,E1 -5560.681,E2 -5560.681} C_VEL
LIN {X 0,Y 509.862,Z 190.97,A -85,B 0,C 180,E1 -5563.174,E2 -5563.174} C_VEL
LIN {X 0,Y 509.855,Z 190.976,A -85,B 0,C 180,E1 -5565.634,E2 -5565.634} C_VEL
LIN {X 0,Y 509.913,Z 190.963,A -85,B 0,C 180,E1 -5568.874,E2 -5568.874} C_VEL
LIN {X 0,Y 509.951,Z 190.962,A -85,B 0,C 180,E1 -5572.078,E2 -5572.078} C_VEL
LIN {X 0,Y 509.979,Z 190.956,A -85,B 0,C 180,E1 -5574.464,E2 -5574.464} C_VEL
LIN {X 0,Y 510.056,Z 190.951,A -85,B 0,C 180,E1 -5577.631,E2 -5577.631} C_VEL
LIN {X 0,Y 510.062,Z 190.948,A -85,B 0,C 180,E1 -5580.789,E2 -5580.789} C_VEL
LIN {X 0,Y 509.953,Z 190.966,A -85,B 0,C 180,E1 -5583.16,E2 -5583.16} C_VEL
LIN {X 0,Y 509.942,Z 190.961,A -85,B 0,C 180,E1 -5586.33,E2 -5586.33} C_VEL
LIN {X 0,Y 509.904,Z 190.969,A -85,B 0,C 180,E1 -5588.72,E2 -5588.72} C_VEL
LIN {X 0,Y 509.905,Z 190.968,A -85,B 0,C 180,E1 -5591.932,E2 -5591.932} C_VEL
LIN {X 0,Y 509.894,Z 190.973,A -85,B 0,C 180,E1 -5595.242,E2 -5595.242} C_VEL
LIN {X 0,Y 509.867,Z 190.972,A -85,B 0,C 180,E1 -5597.993,E2 -5597.993} C_VEL
LIN {X 0,Y 509.901,Z 190.972,A -85,B 0,C 180,E1 -5600.406,E2 -5600.406} C_VEL
LIN {X 0,Y 509.934,Z 191.16,A -85,B 0,C 180,E1 -5601.528,E2 -5601.528} C_VEL
LIN {X 0,Y 510.317,Z 196.236,A -85,B 0,C 180,E1 -5602.478,E2 -5602.478} C_VEL
LIN {X 0,Y 512.33,Z 206.624,A -85,B 0,C 180,E1 -5602.705,E2 -5602.705} C_VEL
LIN {X 0,Y 511.743,Z 302.881,A -85,B 0,C 180,E1 -5604.115,E2 -5604.115} C_VEL
LIN {X 0,Y 511.585,Z 315.898,A -85,B 0,C 180,E1 -5604.46,E2 -5604.46} C_VEL
LIN {X 0,Y 511.354,Z 328.484,A -85,B 0,C 180,E1 -5604.954,E2 -5604.954} C_VEL
LIN {X 0,Y 511.137,Z 339.827,A -85,B 0,C 180,E1 -5605.556,E2 -5605.556} C_VEL
LIN {X 0,Y 510.851,Z 350.188,A -85,B 0,C 180,E1 -5606.258,E2 -5606.258} C_VEL
LIN {X 0,Y 510.502,Z 360.558,A -85,B 0,C 180,E1 -5607.131,E2 -5607.131} C_VEL
LIN {X 0,Y 510.207,Z 370.482,A -85,B 0,C 180,E1 -5608.166,E2 -5608.166} C_VEL
LIN {X 0,Y 509.943,Z 379.166,A -85,B 0,C 180,E1 -5609.292,E2 -5609.292} C_VEL
LIN {X 0,Y 509.728,Z 386.345,A -85,B 0,C 180,E1 -5610.444,E2 -5610.444} C_VEL
LIN {X 0,Y 509.561,Z 393.24,A -85,B 0,C 180,E1 -5611.84,E2 -5611.84} C_VEL
LIN {X 0,Y 509.399,Z 397.876,A -85,B 0,C 180,E1 -5613.06,E2 -5613.06} C_VEL
LIN {X 0,Y 509.282,Z 401.766,A -85,B 0,C 180,E1 -5614.457,E2 -5614.457} C_VEL
LIN {X 0,Y 509.236,Z 403.793,A -85,B 0,C 180,E1 -5615.486,E2 -5615.486} C_VEL
LIN {X 0,Y 509.201,Z 405.368,A -85,B 0,C 180,E1 -5616.821,E2 -5616.821} C_VEL
LIN {X 0,Y 509.17,Z 405.728,A -85,B 0,C 180,E1 -5617.558,E2 -5617.558} C_VEL
LIN {X 0,Y 508.474,Z 405.85,A -85,B 0,C 180,E1 -5618.219,E2 -5618.219} C_VEL
LIN {X 0,Y 505.615,Z 405.582,A -85,B 0,C 180,E1 -5619.292,E2 -5619.292} C_VEL
LIN {X 0,Y 503.237,Z 404.842,A -85,B 0,C 180,E1 -5620.152,E2 -5620.152} C_VEL
LIN {X 0,Y 502.24,Z 403.921,A -85,B 0,C 180,E1 -5620.811,E2 -5620.811} C_VEL
LIN {X 0,Y 502.172,Z 403.522,A -85,B 0,C 180,E1 -5621.032,E2 -5621.032} C_VEL
LIN {X 0,Y 502.276,Z 400.896,A -85,B 0,C 180,E1 -5622.193,E2 -5622.193} C_VEL
LIN {X 0,Y 502.382,Z 397.434,A -85,B 0,C 180,E1 -5623.327,E2 -5623.327} C_VEL
LIN {X 0,Y 502.529,Z 391.967,A -85,B 0,C 180,E1 -5624.692,E2 -5624.692} C_VEL
LIN {X 0,Y 502.66,Z 386.143,A -85,B 0,C 180,E1 -5625.838,E2 -5625.838} C_VEL
LIN {X 0,Y 502.931,Z 378.557,A -85,B 0,C 180,E1 -5627.042,E2 -5627.042} C_VEL
LIN {X 0,Y 503.245,Z 369.669,A -85,B 0,C 180,E1 -5628.174,E2 -5628.174} C_VEL
LIN {X 0,Y 503.624,Z 358.912,A -85,B 0,C 180,E1 -5629.278,E2 -5629.278} C_VEL
LIN {X 0,Y 503.903,Z 347.847,A -85,B 0,C 180,E1 -5630.176,E2 -5630.176} C_VEL
LIN {X 0,Y 504.282,Z 335.386,A -85,B 0,C 180,E1 -5630.968,E2 -5630.968} C_VEL
LIN {X 0,Y 504.591,Z 324.22,A -85,B 0,C 180,E1 -5631.508,E2 -5631.508} C_VEL
LIN {X 0,Y 504.76,Z 311.03,A -85,B 0,C 180,E1 -5631.967,E2 -5631.967} C_VEL
LIN {X 0,Y 504.907,Z 298.516,A -85,B 0,C 180,E1 -5632.244,E2 -5632.244} C_VEL
LIN {X 0,Y 505.442,Z 206.831,A -85,B 0,C 180,E1 -5633.59,E2 -5633.59} C_VEL
LIN {X 0,Y 503.302,Z 196.314,A -85,B 0,C 180,E1 -5633.83,E2 -5633.83} C_VEL
LIN {X 0,Y 502.818,Z 191.854,A -85,B 0,C 180,E1 -5634.791,E2 -5634.791} C_VEL
LIN {X 0,Y 502.782,Z 191.855,A -85,B 0,C 180,E1 -5637.915,E2 -5637.915} C_VEL
LIN {X 0,Y 502.823,Z 191.849,A -85,B 0,C 180,E1 -5640.712,E2 -5640.712} C_VEL
LIN {X 0,Y 502.844,Z 191.848,A -85,B 0,C 180,E1 -5643.444,E2 -5643.444} C_VEL
LIN {X 0,Y 502.787,Z 191.858,A -85,B 0,C 180,E1 -5646.959,E2 -5646.959} C_VEL
LIN {X 0,Y 502.834,Z 191.847,A -85,B 0,C 180,E1 -5649.548,E2 -5649.548} C_VEL
LIN {X 0,Y 502.818,Z 191.847,A -85,B 0,C 180,E1 -5652.092,E2 -5652.092} C_VEL
LIN {X 0,Y 502.841,Z 191.846,A -85,B 0,C 180,E1 -5655.429,E2 -5655.429} C_VEL
LIN {X 0,Y 502.878,Z 191.847,A -85,B 0,C 180,E1 -5658.717,E2 -5658.717} C_VEL
LIN {X 0,Y 502.882,Z 191.84,A -85,B 0,C 180,E1 -5661.967,E2 -5661.967} C_VEL
LIN {X 0,Y 502.93,Z 191.838,A -85,B 0,C 180,E1 -5664.387,E2 -5664.387} C_VEL
LIN {X 0,Y 503.021,Z 191.822,A -85,B 0,C 180,E1 -5667.598,E2 -5667.598} C_VEL
LIN {X 0,Y 503.012,Z 191.827,A -85,B 0,C 180,E1 -5670.801,E2 -5670.801} C_VEL
LIN {X 0,Y 503.019,Z 191.83,A -85,B 0,C 180,E1 -5672.402,E2 -5672.402} C_VEL
LIN {X 0,Y 502.927,Z 191.834,A -85,B 0,C 180,E1 -5675.614,E2 -5675.614} C_VEL
LIN {X 0,Y 502.87,Z 191.842,A -85,B 0,C 180,E1 -5678.844,E2 -5678.844} C_VEL
LIN {X 0,Y 502.847,Z 191.85,A -85,B 0,C 180,E1 -5682.102,E2 -5682.102} C_VEL
LIN {X 0,Y 502.851,Z 191.843,A -85,B 0,C 180,E1 -5685.4,E2 -5685.4} C_VEL
LIN {X 0,Y 502.824,Z 191.847,A -85,B 0,C 180,E1 -5688.752,E2 -5688.752} C_VEL
LIN {X 0,Y 502.783,Z 191.852,A -85,B 0,C 180,E1 -5691.311,E2 -5691.311} C_VEL
LIN {X 0,Y 502.77,Z 191.862,A -85,B 0,C 180,E1 -5693.915,E2 -5693.915} C_VEL
LIN {X 0,Y 502.836,Z 191.845,A -85,B 0,C 180,E1 -5696.568,E2 -5696.568} C_VEL
LIN {X 0,Y 502.816,Z 191.854,A -85,B 0,C 180,E1 -5699.935,E2 -5699.935} C_VEL
LIN {X 0,Y 502.834,Z 191.846,A -85,B 0,C 180,E1 -5703.031,E2 -5703.031} C_VEL
LIN {X 0,Y 502.77,Z 191.857,A -85,B 0,C 180,E1 -5705.952,E2 -5705.952} C_VEL
LIN {X 0,Y 502.795,Z 191.851,A -85,B 0,C 180,E1 -5708.977,E2 -5708.977} C_VEL
LIN {X 0,Y 502.806,Z 191.849,A -85,B 0,C 180,E1 -5712.199,E2 -5712.199} C_VEL
LIN {X 0,Y 502.788,Z 191.859,A -85,B 0,C 180,E1 -5715.47,E2 -5715.47} C_VEL
LIN {X 0,Y 502.797,Z 191.852,A -85,B 0,C 180,E1 -5717.861,E2 -5717.861} C_VEL
LIN {X 0,Y 502.795,Z 191.855,A -85,B 0,C 180,E1 -5721.023,E2 -5721.023} C_VEL
LIN {X 0,Y 502.773,Z 191.852,A -85,B 0,C 180,E1 -5724.17,E2 -5724.17} C_VEL
LIN {X 0,Y 502.833,Z 191.851,A -85,B 0,C 180,E1 -5726.994,E2 -5726.994} C_VEL
LIN {X 0,Y 502.812,Z 191.848,A -85,B 0,C 180,E1 -5730.066,E2 -5730.066} C_VEL
LIN {X 0,Y 502.847,Z 191.846,A -85,B 0,C 180,E1 -5733.444,E2 -5733.444} C_VEL
LIN {X 0,Y 502.789,Z 191.859,A -85,B 0,C 180,E1 -5736.959,E2 -5736.959} C_VEL
LIN {X 0,Y 502.837,Z 191.845,A -85,B 0,C 180,E1 -5739.548,E2 -5739.548} C_VEL
LIN {X 0,Y 502.82,Z 191.847,A -85,B 0,C 180,E1 -5742.092,E2 -5742.092} C_VEL
LIN {X 0,Y 502.83,Z 191.846,A -85,B 0,C 180,E1 -5745.429,E2 -5745.429} C_VEL
LIN {X 0,Y 502.879,Z 191.847,A -85,B 0,C 180,E1 -5748.717,E2 -5748.717} C_VEL
LIN {X 0,Y 502.875,Z 191.841,A -85,B 0,C 180,E1 -5751.966,E2 -5751.966} C_VEL
LIN {X 0,Y 502.918,Z 191.842,A -85,B 0,C 180,E1 -5754.386,E2 -5754.386} C_VEL
LIN {X 0,Y 503.02,Z 191.822,A -85,B 0,C 180,E1 -5757.598,E2 -5757.598} C_VEL
LIN {X 0,Y 502.973,Z 191.83,A -85,B 0,C 180,E1 -5760.801,E2 -5760.801} C_VEL
LIN {X 0,Y 503.014,Z 191.83,A -85,B 0,C 180,E1 -5762.402,E2 -5762.402} C_VEL
LIN {X 0,Y 502.901,Z 191.838,A -85,B 0,C 180,E1 -5765.614,E2 -5765.614} C_VEL
LIN {X 0,Y 502.852,Z 191.849,A -85,B 0,C 180,E1 -5768.034,E2 -5768.034} C_VEL
LIN {X 0,Y 502.879,Z 191.84,A -85,B 0,C 180,E1 -5771.283,E2 -5771.283} C_VEL
LIN {X 0,Y 502.834,Z 191.847,A -85,B 0,C 180,E1 -5774.571,E2 -5774.571} C_VEL
LIN {X 0,Y 502.812,Z 191.854,A -85,B 0,C 180,E1 -5778.109,E2 -5778.109} C_VEL
LIN {X 0,Y 502.833,Z 191.846,A -85,B 0,C 180,E1 -5780.536,E2 -5780.536} C_VEL
LIN {X 0,Y 502.789,Z 191.851,A -85,B 0,C 180,E1 -5783.041,E2 -5783.041} C_VEL
LIN {X 0,Y 502.781,Z 191.859,A -85,B 0,C 180,E1 -5785.679,E2 -5785.679} C_VEL
LIN {X 0,Y 502.776,Z 191.853,A -85,B 0,C 180,E1 -5788.377,E2 -5788.377} C_VEL
LIN {X 0,Y 502.795,Z 191.852,A -85,B 0,C 180,E1 -5791.144,E2 -5791.144} C_VEL
LIN {X 0,Y 502.789,Z 191.853,A -85,B 0,C 180,E1 -5793.995,E2 -5793.995} C_VEL
LIN {X 0,Y 502.767,Z 191.858,A -85,B 0,C 180,E1 -5797.176,E2 -5797.176} C_VEL
LIN {X 0,Y 502.775,Z 191.854,A -85,B 0,C 180,E1 -5800.017,E2 -5800.017} C_VEL
LIN {X 0,Y 502.75,Z 191.863,A -85,B 0,C 180,E1 -5803.234,E2 -5803.234} C_VEL
LIN {X 0,Y 502.781,Z 191.855,A -85,B 0,C 180,E1 -5805.66,E2 -5805.66} C_VEL
LIN {X 0,Y 502.767,Z 191.859,A -85,B 0,C 180,E1 -5809.012,E2 -5809.012} C_VEL
LIN {X 0,Y 502.792,Z 191.85,A -85,B 0,C 180,E1 -5812.046,E2 -5812.046} C_VEL
LIN {X 0,Y 502.794,Z 191.859,A -85,B 0,C 180,E1 -5815.033,E2 -5815.033} C_VEL
LIN {X 0,Y 502.781,Z 191.853,A -85,B 0,C 180,E1 -5817.915,E2 -5817.915} C_VEL
LIN {X 0,Y 502.806,Z 191.856,A -85,B 0,C 180,E1 -5820.711,E2 -5820.711} C_VEL
LIN {X 0,Y 502.838,Z 191.962,A -85,B 0,C 180,E1 -5823.256,E2 -5823.256} C_VEL
LIN {X 0,Y 504.917,Z 202.598,A -85,B 0,C 180,E1 -5824.953,E2 -5824.953} C_VEL
LIN {X 0,Y 504.531,Z 218.248,A -85,B 0,C 180,E1 -5827.26,E2 -5827.26} C_VEL
LIN {X 0,Y 503.967,Z 238.733,A -85,B 0,C 180,E1 -5830.234,E2 -5830.234} C_VEL
LIN {X 0,Y 503.377,Z 260.608,A -85,B 0,C 180,E1 -5833.368,E2 -5833.368} C_VEL
LIN {X 0,Y 503.236,Z 266.414,A -85,B 0,C 180,E1 -5834.19,E2 -5834.19} C_VEL
LIN {X 0,Y 505.293,Z 282.388,A -85,B 0,C 180,E1 -5834.491,E2 -5834.491} C_VEL
LIN {X 0,Y 504.716,Z 375.64,A -85,B 0,C 180,E1 -5835.87,E2 -5835.87} C_VEL
LIN {X 0,Y 504.403,Z 388.822,A -85,B 0,C 180,E1 -5836.221,E2 -5836.221} C_VEL
LIN {X 0,Y 504.128,Z 400.984,A -85,B 0,C 180,E1 -5836.701,E2 -5836.701} C_VEL
LIN {X 0,Y 503.735,Z 412.467,A -85,B 0,C 180,E1 -5837.306,E2 -5837.306} C_VEL
LIN {X 0,Y 503.345,Z 424.282,A -85,B 0,C 180,E1 -5838.115,E2 -5838.115} C_VEL
LIN {X 0,Y 503.063,Z 434.902,A -85,B 0,C 180,E1 -5839.027,E2 -5839.027} C_VEL
LIN {X 0,Y 502.767,Z 443.583,A -85,B 0,C 180,E1 -5839.937,E2 -5839.937} C_VEL
LIN {X 0,Y 502.55,Z 451.594,A -85,B 0,C 180,E1 -5840.948,E2 -5840.948} C_VEL
LIN {X 0,Y 502.365,Z 459.43,A -85,B 0,C 180,E1 -5842.16,E2 -5842.16} C_VEL
LIN {X 0,Y 502.236,Z 466.631,A -85,B 0,C 180,E1 -5843.572,E2 -5843.572} C_VEL
LIN {X 0,Y 502.177,Z 471.427,A -85,B 0,C 180,E1 -5844.78,E2 -5844.78} C_VEL
LIN {X 0,Y 502.207,Z 475.094,A -85,B 0,C 180,E1 -5845.987,E2 -5845.987} C_VEL
LIN {X 0,Y 502.175,Z 476.981,A -85,B 0,C 180,E1 -5846.791,E2 -5846.791} C_VEL
LIN {X 0,Y 502.128,Z 478.394,A -85,B 0,C 180,E1 -5847.593,E2 -5847.593} C_VEL
LIN {X 0,Y 502.035,Z 480.001,A -85,B 0,C 180,E1 -5849.198,E2 -5849.198} C_VEL
LIN {X 0,Y 502.042,Z 480.212,A -85,B 0,C 180,E1 -5850,E2 -5850} C_VEL
LIN {X 0,Y 502.036,Z 479.982,A -85,B 0,C 180,E1 -5850.802,E2 -5850.802} C_VEL
LIN {X 0,Y 502.129,Z 478.332,A -85,B 0,C 180,E1 -5852.406,E2 -5852.406} C_VEL
LIN {X 0,Y 502.188,Z 476.9,A -85,B 0,C 180,E1 -5853.209,E2 -5853.209} C_VEL
LIN {X 0,Y 502.146,Z 473.886,A -85,B 0,C 180,E1 -5854.415,E2 -5854.415} C_VEL
LIN {X 0,Y 502.211,Z 469.819,A -85,B 0,C 180,E1 -5855.621,E2 -5855.621} C_VEL
LIN {X 0,Y 502.291,Z 463.667,A -85,B 0,C 180,E1 -5857.012,E2 -5857.012} C_VEL
LIN {X 0,Y 502.426,Z 456.737,A -85,B 0,C 180,E1 -5858.243,E2 -5858.243} C_VEL
LIN {X 0,Y 502.632,Z 448.275,A -85,B 0,C 180,E1 -5859.456,E2 -5859.456} C_VEL
LIN {X 0,Y 502.897,Z 439.579,A -85,B 0,C 180,E1 -5860.467,E2 -5860.467} C_VEL
LIN {X 0,Y 503.178,Z 428.854,A -85,B 0,C 180,E1 -5861.48,E2 -5861.48} C_VEL
LIN {X 0,Y 503.532,Z 417.355,A -85,B 0,C 180,E1 -5862.352,E2 -5862.352} C_VEL
LIN {X 0,Y 503.915,Z 405.545,A -85,B 0,C 180,E1 -5863.048,E2 -5863.048} C_VEL
LIN {X 0,Y 504.278,Z 393.115,A -85,B 0,C 180,E1 -5863.602,E2 -5863.602} C_VEL
LIN {X 0,Y 504.598,Z 380.4,A -85,B 0,C 180,E1 -5864.004,E2 -5864.004} C_VEL
LIN {X 0,Y 504.8,Z 365.453,A -85,B 0,C 180,E1 -5864.281,E2 -5864.281} C_VEL
LIN {X 0,Y 505.135,Z 280.393,A -85,B 0,C 180,E1 -5865.531,E2 -5865.531} C_VEL
LIN {X 0,Y 503.163,Z 265.249,A -85,B 0,C 180,E1 -5865.843,E2 -5865.843} C_VEL
LIN {X 0,Y 503.685,Z 243.098,A -85,B 0,C 180,E1 -5868.93,E2 -5868.93} C_VEL
LIN {X 0,Y 504.08,Z 222.062,A -85,B 0,C 180,E1 -5871.898,E2 -5871.898} C_VEL
LIN {X 0,Y 504.55,Z 202.351,A -85,B 0,C 180,E1 -5874.7,E2 -5874.7} C_VEL
LIN {X 0,Y 503.68,Z 196.166,A -85,B 0,C 180,E1 -5875.629,E2 -5875.629} C_VEL
LIN {X 0,Y 502.811,Z 191.853,A -85,B 0,C 180,E1 -5876.333,E2 -5876.333} C_VEL
LIN {X 0,Y 502.804,Z 191.858,A -85,B 0,C 180,E1 -5879.289,E2 -5879.289} C_VEL
LIN {X 0,Y 502.779,Z 191.854,A -85,B 0,C 180,E1 -5882.085,E2 -5882.085} C_VEL
LIN {X 0,Y 502.794,Z 191.858,A -85,B 0,C 180,E1 -5884.966,E2 -5884.966} C_VEL
LIN {X 0,Y 502.791,Z 191.856,A -85,B 0,C 180,E1 -5888.485,E2 -5888.485} C_VEL
LIN {X 0,Y 502.778,Z 191.856,A -85,B 0,C 180,E1 -5891.07,E2 -5891.07} C_VEL
LIN {X 0,Y 502.756,Z 191.856,A -85,B 0,C 180,E1 -5893.372,E2 -5893.372} C_VEL
LIN {X 0,Y 502.779,Z 191.852,A -85,B 0,C 180,E1 -5895.66,E2 -5895.66} C_VEL
LIN {X 0,Y 502.795,Z 191.85,A -85,B 0,C 180,E1 -5897.86,E2 -5897.86} C_VEL
LIN {X 0,Y 502.793,Z 191.853,A -85,B 0,C 180,E1 -5901.023,E2 -5901.023} C_VEL
LIN {X 0,Y 502.771,Z 191.86,A -85,B 0,C 180,E1 -5904.169,E2 -5904.169} C_VEL
LIN {X 0,Y 502.833,Z 191.846,A -85,B 0,C 180,E1 -5906.993,E2 -5906.993} C_VEL
LIN {X 0,Y 502.814,Z 191.855,A -85,B 0,C 180,E1 -5910.065,E2 -5910.065} C_VEL
LIN {X 0,Y 502.844,Z 191.844,A -85,B 0,C 180,E1 -5913.444,E2 -5913.444} C_VEL
LIN {X 0,Y 502.787,Z 191.851,A -85,B 0,C 180,E1 -5916.959,E2 -5916.959} C_VEL
LIN {X 0,Y 502.836,Z 191.848,A -85,B 0,C 180,E1 -5919.548,E2 -5919.548} C_VEL
LIN {X 0,Y 502.817,Z 191.851,A -85,B 0,C 180,E1 -5922.091,E2 -5922.091} C_VEL
LIN {X 0,Y 502.833,Z 191.849,A -85,B 0,C 180,E1 -5925.429,E2 -5925.429} C_VEL
LIN {X 0,Y 502.877,Z 191.839,A -85,B 0,C 180,E1 -5928.717,E2 -5928.717} C_VEL
LIN {X 0,Y 502.901,Z 191.841,A -85,B 0,C 180,E1 -5931.967,E2 -5931.967} C_VEL
LIN {X 0,Y 502.933,Z 191.834,A -85,B 0,C 180,E1 -5934.386,E2 -5934.386} C_VEL
LIN {X 0,Y 503.026,Z 191.827,A -85,B 0,C 180,E1 -5937.598,E2 -5937.598} C_VEL
LIN {X 0,Y 503.028,Z 191.823,A -85,B 0,C 180,E1 -5940,E2 -5940} C_VEL
LIN {X 0,Y 503.025,Z 191.823,A -85,B 0,C 180,E1 -5942.402,E2 -5942.402} C_VEL
LIN {X 0,Y 502.931,Z 191.837,A -85,B 0,C 180,E1 -5945.614,E2 -5945.614} C_VEL
LIN {X 0,Y 502.865,Z 191.847,A -85,B 0,C 180,E1 -5948.843,E2 -5948.843} C_VEL
LIN {X 0,Y 502.846,Z 191.847,A -85,B 0,C 180,E1 -5952.102,E2 -5952.102} C_VEL
LIN {X 0,Y 502.849,Z 191.85,A -85,B 0,C 180,E1 -5955.4,E2 -5955.4} C_VEL
LIN {X 0,Y 502.826,Z 191.854,A -85,B 0,C 180,E1 -5958.752,E2 -5958.752} C_VEL
LIN {X 0,Y 502.864,Z 191.9,A -85,B 0,C 180,E1 -5961.361,E2 -5961.361} C_VEL
LIN {X 0,Y 503.361,Z 196.827,A -85,B 0,C 180,E1 -5962.261,E2 -5962.261} C_VEL
LIN {X 0,Y 505.489,Z 206.702,A -85,B 0,C 180,E1 -5962.483,E2 -5962.483} C_VEL
LIN {X 0,Y 504.859,Z 304.242,A -85,B 0,C 180,E1 -5963.946,E2 -5963.946} C_VEL
LIN {X 0,Y 504.684,Z 317.423,A -85,B 0,C 180,E1 -5964.31,E2 -5964.31} C_VEL
LIN {X 0,Y 504.446,Z 329.956,A -85,B 0,C 180,E1 -5964.821,E2 -5964.821} C_VEL
LIN {X 0,Y 504.197,Z 341.27,A -85,B 0,C 180,E1 -5965.446,E2 -5965.446} C_VEL
LIN {X 0,Y 503.808,Z 353.15,A -85,B 0,C 180,E1 -5966.289,E2 -5966.289} C_VEL
LIN {X 0,Y 503.47,Z 363.703,A -85,B 0,C 180,E1 -5967.235,E2 -5967.235} C_VEL
LIN {X 0,Y 503.162,Z 373.622,A -85,B 0,C 180,E1 -5968.353,E2 -5968.353} C_VEL
LIN {X 0,Y 502.884,Z 381.491,A -85,B 0,C 180,E1 -5969.443,E2 -5969.443} C_VEL
LIN {X 0,Y 502.639,Z 388.758,A -85,B 0,C 180,E1 -5970.687,E2 -5970.687} C_VEL
LIN {X 0,Y 502.452,Z 395.189,A -85,B 0,C 180,E1 -5972.108,E2 -5972.108} C_VEL
LIN {X 0,Y 502.3,Z 400.107,A -85,B 0,C 180,E1 -5973.55,E2 -5973.55} C_VEL
LIN {X 0,Y 502.183,Z 403.549,A -85,B 0,C 180,E1 -5975.015,E2 -5975.015} C_VEL
LIN {X 0,Y 502.132,Z 405.091,A -85,B 0,C 180,E1 -5976.004,E2 -5976.004} C_VEL
LIN {X 0,Y 502.108,Z 406.05,A -85,B 0,C 180,E1 -5977.077,E2 -5977.077} C_VEL
LIN {X 0,Y 502.068,Z 406.282,A -85,B 0,C 180,E1 -5978.382,E2 -5978.382} C_VEL
LIN {X 0,Y 502.102,Z 405.494,A -85,B 0,C 180,E1 -5979.66,E2 -5979.66} C_VEL
LIN {X 0,Y 502.172,Z 403.522,A -85,B 0,C 180,E1 -5981.032,E2 -5981.032} C_VEL
LIN {X 0,Y 501.545,Z 402.238,A -85,B 0,C 180,E1 -5981.687,E2 -5981.687} C_VEL
LIN {X 0,Y 498.749,Z 399.704,A -85,B 0,C 180,E1 -5982.738,E2 -5982.738} C_VEL
LIN {X 0,Y 496.412,Z 397.238,A -85,B 0,C 180,E1 -5983.567,E2 -5983.567} C_VEL
LIN {X 0,Y 495.462,Z 394.979,A -85,B 0,C 180,E1 -5984.193,E2 -5984.193} C_VEL
LIN {X 0,Y 495.416,Z 394.139,A -85,B 0,C 180,E1 -5984.402,E2 -5984.402} C_VEL
LIN {X 0,Y 495.595,Z 387.507,A -85,B 0,C 180,E1 -5985.784,E2 -5985.784} C_VEL
LIN {X 0,Y 495.859,Z 380.614,A -85,B 0,C 180,E1 -5986.93,E2 -5986.93} C_VEL
LIN {X 0,Y 496.194,Z 372.207,A -85,B 0,C 180,E1 -5988.069,E2 -5988.069} C_VEL
LIN {X 0,Y 496.517,Z 362.767,A -85,B 0,C 180,E1 -5989.107,E2 -5989.107} C_VEL
LIN {X 0,Y 496.861,Z 351.442,A -85,B 0,C 180,E1 -5990.105,E2 -5990.105} C_VEL
LIN {X 0,Y 497.275,Z 340.535,A -85,B 0,C 180,E1 -5990.867,E2 -5990.867} C_VEL
LIN {X 0,Y 497.605,Z 328.321,A -85,B 0,C 180,E1 -5991.525,E2 -5991.525} C_VEL
LIN {X 0,Y 497.799,Z 314.756,A -85,B 0,C 180,E1 -5992.06,E2 -5992.06} C_VEL
LIN {X 0,Y 498.005,Z 301.814,A -85,B 0,C 180,E1 -5992.387,E2 -5992.387} C_VEL
LIN {X 0,Y 498.506,Z 206.972,A -85,B 0,C 180,E1 -5993.815,E2 -5993.815} C_VEL
LIN {X 0,Y 496.311,Z 196.727,A -85,B 0,C 180,E1 -5994.052,E2 -5994.052} C_VEL
LIN {X 0,Y 495.777,Z 192.732,A -85,B 0,C 180,E1 -5994.923,E2 -5994.923} C_VEL
LIN {X 0,Y 495.766,Z 192.734,A -85,B 0,C 180,E1 -5997.406,E2 -5997.406} C_VEL
LIN {X 0,Y 495.766,Z 192.725,A -85,B 0,C 180,E1 -6000.254,E2 -6000.254} C_VEL
LIN {X 0,Y 495.805,Z 192.728,A -85,B 0,C 180,E1 -6003.256,E2 -6003.256} C_VEL
LIN {X 0,Y 495.74,Z 192.731,A -85,B 0,C 180,E1 -6006.613,E2 -6006.613} C_VEL
LIN {X 0,Y 495.78,Z 192.728,A -85,B 0,C 180,E1 -6009.324,E2 -6009.324} C_VEL
LIN {X 0,Y 495.78,Z 192.724,A -85,B 0,C 180,E1 -6011.829,E2 -6011.829} C_VEL
LIN {X 0,Y 495.825,Z 192.722,A -85,B 0,C 180,E1 -6014.549,E2 -6014.549} C_VEL
LIN {X 0,Y 495.83,Z 192.718,A -85,B 0,C 180,E1 -6017.966,E2 -6017.966} C_VEL
LIN {X 0,Y 495.835,Z 192.721,A -85,B 0,C 180,E1 -6021.03,E2 -6021.03} C_VEL
LIN {X 0,Y 495.885,Z 192.715,A -85,B 0,C 180,E1 -6024.307,E2 -6024.307} C_VEL
LIN {X 0,Y 495.989,Z 192.698,A -85,B 0,C 180,E1 -6027.564,E2 -6027.564} C_VEL
LIN {X 0,Y 495.963,Z 192.705,A -85,B 0,C 180,E1 -6030.812,E2 -6030.812} C_VEL
LIN {X 0,Y 495.987,Z 192.707,A -85,B 0,C 180,E1 -6032.437,E2 -6032.437} C_VEL
LIN {X 0,Y 495.882,Z 192.712,A -85,B 0,C 180,E1 -6035.694,E2 -6035.694} C_VEL
LIN {X 0,Y 495.839,Z 192.717,A -85,B 0,C 180,E1 -6038.97,E2 -6038.97} C_VEL
LIN {X 0,Y 495.831,Z 192.723,A -85,B 0,C 180,E1 -6042.035,E2 -6042.035} C_VEL
LIN {X 0,Y 495.826,Z 192.719,A -85,B 0,C 180,E1 -6045.451,E2 -6045.451} C_VEL
LIN {X 0,Y 495.78,Z 192.724,A -85,B 0,C 180,E1 -6049.029,E2 -6049.029} C_VEL
LIN {X 0,Y 495.743,Z 192.732,A -85,B 0,C 180,E1 -6051.629,E2 -6051.629} C_VEL
LIN {X 0,Y 495.716,Z 192.735,A -85,B 0,C 180,E1 -6054.277,E2 -6054.277} C_VEL
LIN {X 0,Y 495.76,Z 192.726,A -85,B 0,C 180,E1 -6056.978,E2 -6056.978} C_VEL
LIN {X 0,Y 495.765,Z 192.729,A -85,B 0,C 180,E1 -6060.147,E2 -6060.147} C_VEL
LIN {X 0,Y 495.795,Z 192.724,A -85,B 0,C 180,E1 -6063.245,E2 -6063.245} C_VEL
LIN {X 0,Y 495.714,Z 192.735,A -85,B 0,C 180,E1 -6066.087,E2 -6066.087} C_VEL
LIN {X 0,Y 495.76,Z 192.726,A -85,B 0,C 180,E1 -6068.768,E2 -6068.768} C_VEL
LIN {X 0,Y 495.747,Z 192.733,A -85,B 0,C 180,E1 -6071.783,E2 -6071.783} C_VEL
LIN {X 0,Y 495.739,Z 192.733,A -85,B 0,C 180,E1 -6075.141,E2 -6075.141} C_VEL
LIN {X 0,Y 495.747,Z 192.728,A -85,B 0,C 180,E1 -6078.218,E2 -6078.218} C_VEL
LIN {X 0,Y 495.748,Z 192.734,A -85,B 0,C 180,E1 -6081.408,E2 -6081.408} C_VEL
LIN {X 0,Y 495.747,Z 192.728,A -85,B 0,C 180,E1 -6084.462,E2 -6084.462} C_VEL
LIN {X 0,Y 495.768,Z 192.73,A -85,B 0,C 180,E1 -6087.406,E2 -6087.406} C_VEL
LIN {X 0,Y 495.76,Z 192.726,A -85,B 0,C 180,E1 -6090.253,E2 -6090.253} C_VEL
LIN {X 0,Y 495.776,Z 192.729,A -85,B 0,C 180,E1 -6093.263,E2 -6093.263} C_VEL
LIN {X 0,Y 495.742,Z 192.733,A -85,B 0,C 180,E1 -6096.612,E2 -6096.612} C_VEL
LIN {X 0,Y 495.782,Z 192.726,A -85,B 0,C 180,E1 -6099.324,E2 -6099.324} C_VEL
LIN {X 0,Y 495.782,Z 192.723,A -85,B 0,C 180,E1 -6101.828,E2 -6101.828} C_VEL
LIN {X 0,Y 495.781,Z 192.726,A -85,B 0,C 180,E1 -6105.217,E2 -6105.217} C_VEL
LIN {X 0,Y 495.854,Z 192.722,A -85,B 0,C 180,E1 -6108.555,E2 -6108.555} C_VEL
LIN {X 0,Y 495.833,Z 192.718,A -85,B 0,C 180,E1 -6111.851,E2 -6111.851} C_VEL
LIN {X 0,Y 495.832,Z 192.718,A -85,B 0,C 180,E1 -6115.121,E2 -6115.121} C_VEL
LIN {X 0,Y 495.988,Z 192.698,A -85,B 0,C 180,E1 -6117.564,E2 -6117.564} C_VEL
LIN {X 0,Y 495.925,Z 192.708,A -85,B 0,C 180,E1 -6120.812,E2 -6120.812} C_VEL
LIN {X 0,Y 495.981,Z 192.705,A -85,B 0,C 180,E1 -6122.436,E2 -6122.436} C_VEL
LIN {X 0,Y 495.858,Z 192.716,A -85,B 0,C 180,E1 -6125.694,E2 -6125.694} C_VEL
LIN {X 0,Y 495.817,Z 192.728,A -85,B 0,C 180,E1 -6128.149,E2 -6128.149} C_VEL
LIN {X 0,Y 495.854,Z 192.715,A -85,B 0,C 180,E1 -6131.445,E2 -6131.445} C_VEL
LIN {X 0,Y 495.783,Z 192.724,A -85,B 0,C 180,E1 -6134.783,E2 -6134.783} C_VEL
LIN {X 0,Y 495.775,Z 192.729,A -85,B 0,C 180,E1 -6138.235,E2 -6138.235} C_VEL
LIN {X 0,Y 495.777,Z 192.724,A -85,B 0,C 180,E1 -6140.756,E2 -6140.756} C_VEL
LIN {X 0,Y 495.742,Z 192.731,A -85,B 0,C 180,E1 -6143.388,E2 -6143.388} C_VEL
LIN {X 0,Y 495.742,Z 192.728,A -85,B 0,C 180,E1 -6146.73,E2 -6146.73} C_VEL
LIN {X 0,Y 495.76,Z 192.733,A -85,B 0,C 180,E1 -6149.747,E2 -6149.747} C_VEL
LIN {X 0,Y 495.755,Z 192.727,A -85,B 0,C 180,E1 -6152.595,E2 -6152.595} C_VEL
LIN {X 0,Y 495.745,Z 192.737,A -85,B 0,C 180,E1 -6155.538,E2 -6155.538} C_VEL
LIN {X 0,Y 495.762,Z 192.727,A -85,B 0,C 180,E1 -6158.767,E2 -6158.767} C_VEL
LIN {X 0,Y 495.726,Z 192.733,A -85,B 0,C 180,E1 -6161.784,E2 -6161.784} C_VEL
LIN {X 0,Y 495.74,Z 192.735,A -85,B 0,C 180,E1 -6165.141,E2 -6165.141} C_VEL
LIN {X 0,Y 495.726,Z 192.73,A -85,B 0,C 180,E1 -6168.215,E2 -6168.215} C_VEL
LIN {X 0,Y 495.748,Z 192.732,A -85,B 0,C 180,E1 -6171.408,E2 -6171.408} C_VEL
LIN {X 0,Y 495.745,Z 192.729,A -85,B 0,C 180,E1 -6174.462,E2 -6174.462} C_VEL
LIN {X 0,Y 495.753,Z 192.732,A -85,B 0,C 180,E1 -6177.404,E2 -6177.404} C_VEL
LIN {X 0,Y 495.759,Z 192.729,A -85,B 0,C 180,E1 -6180.253,E2 -6180.253} C_VEL
LIN {X 0,Y 495.82,Z 192.908,A -85,B 0,C 180,E1 -6183.07,E2 -6183.07} C_VEL
LIN {X 0,Y 498.037,Z 204.562,A -85,B 0,C 180,E1 -6184.954,E2 -6184.954} C_VEL
LIN {X 0,Y 497.487,Z 222.156,A -85,B 0,C 180,E1 -6187.578,E2 -6187.578} C_VEL
LIN {X 0,Y 496.838,Z 244.085,A -85,B 0,C 180,E1 -6190.799,E2 -6190.799} C_VEL
LIN {X 0,Y 496.245,Z 265.982,A -85,B 0,C 180,E1 -6193.964,E2 -6193.964} C_VEL
LIN {X 0,Y 498.432,Z 283.662,A -85,B 0,C 180,E1 -6194.303,E2 -6194.303} C_VEL
LIN {X 0,Y 497.792,Z 375.946,A -85,B 0,C 180,E1 -6195.695,E2 -6195.695} C_VEL
LIN {X 0,Y 497.456,Z 389.622,A -85,B 0,C 180,E1 -6196.077,E2 -6196.077} C_VEL
LIN {X 0,Y 497.11,Z 402.485,A -85,B 0,C 180,E1 -6196.614,E2 -6196.614} C_VEL
LIN {X 0,Y 496.698,Z 413.943,A -85,B 0,C 180,E1 -6197.258,E2 -6197.258} C_VEL
LIN {X 0,Y 496.305,Z 424.994,A -85,B 0,C 180,E1 -6198.047,E2 -6198.047} C_VEL
LIN {X 0,Y 496.01,Z 435.409,A -85,B 0,C 180,E1 -6198.972,E2 -6198.972} C_VEL
LIN {X 0,Y 495.669,Z 444.755,A -85,B 0,C 180,E1 -6199.997,E2 -6199.997} C_VEL
LIN {X 0,Y 495.408,Z 453.838,A -85,B 0,C 180,E1 -6201.228,E2 -6201.228} C_VEL
LIN {X 0,Y 495.242,Z 461.158,A -85,B 0,C 180,E1 -6202.457,E2 -6202.457} C_VEL
LIN {X 0,Y 495.117,Z 467.344,A -85,B 0,C 180,E1 -6203.767,E2 -6203.767} C_VEL
LIN {X 0,Y 495.038,Z 472.237,A -85,B 0,C 180,E1 -6205.113,E2 -6205.113} C_VEL
LIN {X 0,Y 495.099,Z 474.572,A -85,B 0,C 180,E1 -6205.93,E2 -6205.93} C_VEL
LIN {X 0,Y 495.095,Z 476.463,A -85,B 0,C 180,E1 -6206.745,E2 -6206.745} C_VEL
LIN {X 0,Y 495.063,Z 477.878,A -85,B 0,C 180,E1 -6207.559,E2 -6207.559} C_VEL
LIN {X 0,Y 494.953,Z 479.482,A -85,B 0,C 180,E1 -6209.186,E2 -6209.186} C_VEL
LIN {X 0,Y 494.962,Z 479.692,A -85,B 0,C 180,E1 -6210,E2 -6210} C_VEL
LIN {X 0,Y 494.955,Z 479.459,A -85,B 0,C 180,E1 -6210.813,E2 -6210.813} C_VEL
LIN {X 0,Y 495.064,Z 477.802,A -85,B 0,C 180,E1 -6212.441,E2 -6212.441} C_VEL
LIN {X 0,Y 495.108,Z 476.365,A -85,B 0,C 180,E1 -6213.255,E2 -6213.255} C_VEL
LIN {X 0,Y 495.045,Z 473.341,A -85,B 0,C 180,E1 -6214.478,E2 -6214.478} C_VEL
LIN {X 0,Y 495.125,Z 469.265,A -85,B 0,C 180,E1 -6215.702,E2 -6215.702} C_VEL
LIN {X 0,Y 495.239,Z 462.995,A -85,B 0,C 180,E1 -6217.133,E2 -6217.133} C_VEL
LIN {X 0,Y 495.347,Z 456.153,A -85,B 0,C 180,E1 -6218.362,E2 -6218.362} C_VEL
LIN {X 0,Y 495.549,Z 447.674,A -85,B 0,C 180,E1 -6219.592,E2 -6219.592} C_VEL
LIN {X 0,Y 495.853,Z 438.962,A -85,B 0,C 180,E1 -6220.618,E2 -6220.618} C_VEL
LIN {X 0,Y 496.193,Z 428.223,A -85,B 0,C 180,E1 -6221.644,E2 -6221.644} C_VEL
LIN {X 0,Y 496.552,Z 416.792,A -85,B 0,C 180,E1 -6222.522,E2 -6222.522} C_VEL
LIN {X 0,Y 496.954,Z 404.851,A -85,B 0,C 180,E1 -6223.234,E2 -6223.234} C_VEL
LIN {X 0,Y 497.336,Z 392.382,A -85,B 0,C 180,E1 -6223.796,E2 -6223.796} C_VEL
LIN {X 0,Y 497.717,Z 379.598,A -85,B 0,C 180,E1 -6224.202,E2 -6224.202} C_VEL
LIN {X 0,Y 497.917,Z 364.515,A -85,B 0,C 180,E1 -6224.483,E2 -6224.483} C_VEL
LIN {X 0,Y 498.315,Z 281.471,A -85,B 0,C 180,E1 -6225.726,E2 -6225.726} C_VEL
LIN {X 0,Y 496.161,Z 264.62,A -85,B 0,C 180,E1 -6226.076,E2 -6226.076} C_VEL
LIN {X 0,Y 496.676,Z 242.541,A -85,B 0,C 180,E1 -6229.207,E2 -6229.207} C_VEL
LIN {X 0,Y 497.11,Z 222.949,A -85,B 0,C 180,E1 -6232.002,E2 -6232.002} C_VEL
LIN {X 0,Y 497.59,Z 203.235,A -85,B 0,C 180,E1 -6234.846,E2 -6234.846} C_VEL
LIN {X 0,Y 496.614,Z 196.974,A -85,B 0,C 180,E1 -6235.805,E2 -6235.805} C_VEL
LIN {X 0,Y 495.786,Z 192.729,A -85,B 0,C 180,E1 -6236.469,E2 -6236.469} C_VEL
LIN {X 0,Y 495.757,Z 192.732,A -85,B 0,C 180,E1 -6239.747,E2 -6239.747} C_VEL
LIN {X 0,Y 495.765,Z 192.732,A -85,B 0,C 180,E1 -6242.594,E2 -6242.594} C_VEL
LIN {X 0,Y 495.745,Z 192.73,A -85,B 0,C 180,E1 -6245.538,E2 -6245.538} C_VEL
LIN {X 0,Y 495.758,Z 192.734,A -85,B 0,C 180,E1 -6248.767,E2 -6248.767} C_VEL
LIN {X 0,Y 495.745,Z 192.729,A -85,B 0,C 180,E1 -6251.782,E2 -6251.782} C_VEL
LIN {X 0,Y 495.737,Z 192.731,A -85,B 0,C 180,E1 -6255.141,E2 -6255.141} C_VEL
LIN {X 0,Y 495.745,Z 192.731,A -85,B 0,C 180,E1 -6258.217,E2 -6258.217} C_VEL
LIN {X 0,Y 495.746,Z 192.729,A -85,B 0,C 180,E1 -6261.408,E2 -6261.408} C_VEL
LIN {X 0,Y 495.745,Z 192.734,A -85,B 0,C 180,E1 -6264.462,E2 -6264.462} C_VEL
LIN {X 0,Y 495.768,Z 192.725,A -85,B 0,C 180,E1 -6267.405,E2 -6267.405} C_VEL
LIN {X 0,Y 495.762,Z 192.731,A -85,B 0,C 180,E1 -6270.253,E2 -6270.253} C_VEL
LIN {X 0,Y 495.774,Z 192.724,A -85,B 0,C 180,E1 -6273.262,E2 -6273.262} C_VEL
LIN {X 0,Y 495.74,Z 192.73,A -85,B 0,C 180,E1 -6276.612,E2 -6276.612} C_VEL
LIN {X 0,Y 495.779,Z 192.725,A -85,B 0,C 180,E1 -6279.324,E2 -6279.324} C_VEL
LIN {X 0,Y 495.779,Z 192.731,A -85,B 0,C 180,E1 -6281.828,E2 -6281.828} C_VEL
LIN {X 0,Y 495.824,Z 192.719,A -85,B 0,C 180,E1 -6284.549,E2 -6284.549} C_VEL
LIN {X 0,Y 495.829,Z 192.721,A -85,B 0,C 180,E1 -6287.965,E2 -6287.965} C_VEL
LIN {X 0,Y 495.838,Z 192.718,A -85,B 0,C 180,E1 -6291.03,E2 -6291.03} C_VEL
LIN {X 0,Y 495.861,Z 192.72,A -85,B 0,C 180,E1 -6293.489,E2 -6293.489} C_VEL
LIN {X 0,Y 495.838,Z 192.717,A -85,B 0,C 180,E1 -6296.75,E2 -6296.75} C_VEL
LIN {X 0,Y 495.867,Z 192.713,A -85,B 0,C 180,E1 -6298.376,E2 -6298.376} C_VEL
LIN {X 0,Y 495.983,Z 192.702,A -85,B 0,C 180,E1 -6300.812,E2 -6300.812} C_VEL
LIN {X 0,Y 495.993,Z 192.699,A -85,B 0,C 180,E1 -6302.436,E2 -6302.436} C_VEL
LIN {X 0,Y 495.886,Z 192.714,A -85,B 0,C 180,E1 -6305.694,E2 -6305.694} C_VEL
LIN {X 0,Y 495.835,Z 192.725,A -85,B 0,C 180,E1 -6308.97,E2 -6308.97} C_VEL
LIN {X 0,Y 495.829,Z 192.722,A -85,B 0,C 180,E1 -6312.035,E2 -6312.035} C_VEL
LIN {X 0,Y 495.824,Z 192.724,A -85,B 0,C 180,E1 -6315.452,E2 -6315.452} C_VEL
LIN {X 0,Y 495.779,Z 192.728,A -85,B 0,C 180,E1 -6318.237,E2 -6318.237} C_VEL
LIN {X 0,Y 495.815,Z 192.77,A -85,B 0,C 180,E1 -6321.189,E2 -6321.189} C_VEL
LIN {X 0,Y 496.386,Z 197.152,A -85,B 0,C 180,E1 -6322.009,E2 -6322.009} C_VEL
LIN {X 0,Y 498.74,Z 208.369,A -85,B 0,C 180,E1 -6322.281,E2 -6322.281} C_VEL
LIN {X 0,Y 497.985,Z 304.865,A -85,B 0,C 180,E1 -6323.753,E2 -6323.753} C_VEL
LIN {X 0,Y 497.808,Z 317.963,A -85,B 0,C 180,E1 -6324.12,E2 -6324.12} C_VEL
LIN {X 0,Y 497.566,Z 330.208,A -85,B 0,C 180,E1 -6324.625,E2 -6324.625} C_VEL
LIN {X 0,Y 497.309,Z 341.476,A -85,B 0,C 180,E1 -6325.251,E2 -6325.251} C_VEL
LIN {X 0,Y 496.942,Z 352.126,A -85,B 0,C 180,E1 -6326.003,E2 -6326.003} C_VEL
LIN {X 0,Y 496.584,Z 362.631,A -85,B 0,C 180,E1 -6326.929,E2 -6326.929} C_VEL
LIN {X 0,Y 496.276,Z 371.257,A -85,B 0,C 180,E1 -6327.861,E2 -6327.861} C_VEL
LIN {X 0,Y 495.941,Z 380.135,A -85,B 0,C 180,E1 -6329.036,E2 -6329.036} C_VEL
LIN {X 0,Y 495.663,Z 388.188,A -85,B 0,C 180,E1 -6330.379,E2 -6330.379} C_VEL
LIN {X 0,Y 495.504,Z 394.339,A -85,B 0,C 180,E1 -6331.678,E2 -6331.678} C_VEL
LIN {X 0,Y 495.258,Z 399.626,A -85,B 0,C 180,E1 -6333.15,E2 -6333.15} C_VEL
LIN {X 0,Y 495.127,Z 403.333,A -85,B 0,C 180,E1 -6334.595,E2 -6334.595} C_VEL
LIN {X 0,Y 495.067,Z 405.629,A -85,B 0,C 180,E1 -6335.985,E2 -6335.985} C_VEL
LIN {X 0,Y 495.009,Z 406.802,A -85,B 0,C 180,E1 -6337.626,E2 -6337.626} C_VEL
LIN {X 0,Y 495.012,Z 406.741,A -85,B 0,C 180,E1 -6338.66,E2 -6338.66} C_VEL
LIN {X 0,Y 495.04,Z 405.744,A -85,B 0,C 180,E1 -6339.948,E2 -6339.948} C_VEL
LIN {X 0,Y 495.124,Z 403.787,A -85,B 0,C 180,E1 -6341.21,E2 -6341.21} C_VEL
LIN {X 0,Y 495.232,Z 400.898,A -85,B 0,C 180,E1 -6342.443,E2 -6342.443} C_VEL
LIN {X 0,Y 495.324,Z 397.082,A -85,B 0,C 180,E1 -6343.646,E2 -6343.646} C_VEL
LIN {X 0,Y 495.416,Z 394.139,A -85,B 0,C 180,E1 -6344.402,E2 -6344.402} C_VEL
LIN {X 0,Y 494.86,Z 391.583,A -85,B 0,C 180,E1 -6345.015,E2 -6345.015} C_VEL
LIN {X 0,Y 492.176,Z 387.044,A -85,B 0,C 180,E1 -6345.992,E2 -6345.992} C_VEL
LIN {X 0,Y 489.508,Z 381.829,A -85,B 0,C 180,E1 -6346.929,E2 -6346.929} C_VEL
LIN {X 0,Y 488.982,Z 378.214,A -85,B 0,C 180,E1 -6347.475,E2 -6347.475} C_VEL
LIN {X 0,Y 489.36,Z 368.924,A -85,B 0,C 180,E1 -6348.652,E2 -6348.652} C_VEL
LIN {X 0,Y 489.716,Z 359.664,A -85,B 0,C 180,E1 -6349.605,E2 -6349.605} C_VEL
LIN {X 0,Y 490.029,Z 349.903,A -85,B 0,C 180,E1 -6350.426,E2 -6350.426} C_VEL
LIN {X 0,Y 490.433,Z 337.667,A -85,B 0,C 180,E1 -6351.241,E2 -6351.241} C_VEL
LIN {X 0,Y 490.823,Z 325.034,A -85,B 0,C 180,E1 -6351.88,E2 -6351.88} C_VEL
LIN {X 0,Y 490.987,Z 312.355,A -85,B 0,C 180,E1 -6352.336,E2 -6352.336} C_VEL
LIN {X 0,Y 491.126,Z 299.517,A -85,B 0,C 180,E1 -6352.631,E2 -6352.631} C_VEL
LIN {X 0,Y 491.781,Z 208.452,A -85,B 0,C 180,E1 -6354.016,E2 -6354.016} C_VEL
LIN {X 0,Y 489.295,Z 197.051,A -85,B 0,C 180,E1 -6354.302,E2 -6354.302} C_VEL
LIN {X 0,Y 488.756,Z 193.607,A -85,B 0,C 180,E1 -6355.047,E2 -6355.047} C_VEL
LIN {X 0,Y 488.703,Z 193.608,A -85,B 0,C 180,E1 -6358.046,E2 -6358.046} C_VEL
LIN {X 0,Y 488.722,Z 193.606,A -85,B 0,C 180,E1 -6360.73,E2 -6360.73} C_VEL
LIN {X 0,Y 488.732,Z 193.605,A -85,B 0,C 180,E1 -6363.527,E2 -6363.527} C_VEL
LIN {X 0,Y 488.708,Z 193.612,A -85,B 0,C 180,E1 -6366.98,E2 -6366.98} C_VEL
LIN {X 0,Y 488.724,Z 193.603,A -85,B 0,C 180,E1 -6369.811,E2 -6369.811} C_VEL
LIN {X 0,Y 488.71,Z 193.607,A -85,B 0,C 180,E1 -6372.423,E2 -6372.423} C_VEL
LIN {X 0,Y 488.761,Z 193.605,A -85,B 0,C 180,E1 -6375,E2 -6375} C_VEL
LIN {X 0,Y 488.807,Z 193.596,A -85,B 0,C 180,E1 -6378.388,E2 -6378.388} C_VEL
LIN {X 0,Y 488.786,Z 193.595,A -85,B 0,C 180,E1 -6381.733,E2 -6381.733} C_VEL
LIN {X 0,Y 488.842,Z 193.591,A -85,B 0,C 180,E1 -6384.224,E2 -6384.224} C_VEL
LIN {X 0,Y 488.956,Z 193.574,A -85,B 0,C 180,E1 -6387.529,E2 -6387.529} C_VEL
LIN {X 0,Y 488.915,Z 193.583,A -85,B 0,C 180,E1 -6390.824,E2 -6390.824} C_VEL
LIN {X 0,Y 488.953,Z 193.582,A -85,B 0,C 180,E1 -6392.472,E2 -6392.472} C_VEL
LIN {X 0,Y 488.84,Z 193.59,A -85,B 0,C 180,E1 -6395.776,E2 -6395.776} C_VEL
LIN {X 0,Y 488.788,Z 193.603,A -85,B 0,C 180,E1 -6398.267,E2 -6398.267} C_VEL
LIN {X 0,Y 488.807,Z 193.594,A -85,B 0,C 180,E1 -6401.613,E2 -6401.613} C_VEL
LIN {X 0,Y 488.759,Z 193.598,A -85,B 0,C 180,E1 -6405.001,E2 -6405.001} C_VEL
LIN {X 0,Y 488.747,Z 193.603,A -85,B 0,C 180,E1 -6408.443,E2 -6408.443} C_VEL
LIN {X 0,Y 488.709,Z 193.605,A -85,B 0,C 180,E1 -6411.071,E2 -6411.071} C_VEL
LIN {X 0,Y 488.672,Z 193.615,A -85,B 0,C 180,E1 -6413.747,E2 -6413.747} C_VEL
LIN {X 0,Y 488.726,Z 193.602,A -85,B 0,C 180,E1 -6416.928,E2 -6416.928} C_VEL
LIN {X 0,Y 488.724,Z 193.605,A -85,B 0,C 180,E1 -6420.22,E2 -6420.22} C_VEL
LIN {X 0,Y 488.737,Z 193.606,A -85,B 0,C 180,E1 -6423.484,E2 -6423.484} C_VEL
LIN {X 0,Y 488.675,Z 193.609,A -85,B 0,C 180,E1 -6426.353,E2 -6426.353} C_VEL
LIN {X 0,Y 488.696,Z 193.61,A -85,B 0,C 180,E1 -6429.255,E2 -6429.255} C_VEL
LIN {X 0,Y 488.69,Z 193.607,A -85,B 0,C 180,E1 -6432.526,E2 -6432.526} C_VEL
LIN {X 0,Y 488.703,Z 193.61,A -85,B 0,C 180,E1 -6435.197,E2 -6435.197} C_VEL
LIN {X 0,Y 488.682,Z 193.608,A -85,B 0,C 180,E1 -6438.582,E2 -6438.582} C_VEL
LIN {X 0,Y 488.679,Z 193.61,A -85,B 0,C 180,E1 -6441.8,E2 -6441.8} C_VEL
LIN {X 0,Y 488.721,Z 193.609,A -85,B 0,C 180,E1 -6445.053,E2 -6445.053} C_VEL
LIN {X 0,Y 488.705,Z 193.605,A -85,B 0,C 180,E1 -6448.046,E2 -6448.046} C_VEL
LIN {X 0,Y 488.704,Z 193.609,A -85,B 0,C 180,E1 -6450.728,E2 -6450.728} C_VEL
LIN {X 0,Y 488.718,Z 193.605,A -85,B 0,C 180,E1 -6453.526,E2 -6453.526} C_VEL
LIN {X 0,Y 488.672,Z 193.61,A -85,B 0,C 180,E1 -6456.253,E2 -6456.253} C_VEL
LIN {X 0,Y 488.75,Z 193.604,A -85,B 0,C 180,E1 -6459.176,E2 -6459.176} C_VEL
LIN {X 0,Y 488.751,Z 193.6,A -85,B 0,C 180,E1 -6461.632,E2 -6461.632} C_VEL
LIN {X 0,Y 488.757,Z 193.603,A -85,B 0,C 180,E1 -6464.999,E2 -6464.999} C_VEL
LIN {X 0,Y 488.809,Z 193.597,A -85,B 0,C 180,E1 -6468.388,E2 -6468.388} C_VEL
LIN {X 0,Y 488.783,Z 193.596,A -85,B 0,C 180,E1 -6471.733,E2 -6471.733} C_VEL
LIN {X 0,Y 488.831,Z 193.594,A -85,B 0,C 180,E1 -6474.224,E2 -6474.224} C_VEL
LIN {X 0,Y 488.955,Z 193.574,A -85,B 0,C 180,E1 -6477.529,E2 -6477.529} C_VEL
LIN {X 0,Y 488.948,Z 193.578,A -85,B 0,C 180,E1 -6480,E2 -6480} C_VEL
LIN {X 0,Y 488.947,Z 193.581,A -85,B 0,C 180,E1 -6482.471,E2 -6482.471} C_VEL
LIN {X 0,Y 488.818,Z 193.594,A -85,B 0,C 180,E1 -6485.776,E2 -6485.776} C_VEL
LIN {X 0,Y 488.765,Z 193.605,A -85,B 0,C 180,E1 -6488.267,E2 -6488.267} C_VEL
LIN {X 0,Y 488.809,Z 193.595,A -85,B 0,C 180,E1 -6491.612,E2 -6491.612} C_VEL
LIN {X 0,Y 488.752,Z 193.599,A -85,B 0,C 180,E1 -6495.001,E2 -6495.001} C_VEL
LIN {X 0,Y 488.747,Z 193.602,A -85,B 0,C 180,E1 -6498.443,E2 -6498.443} C_VEL
LIN {X 0,Y 488.709,Z 193.605,A -85,B 0,C 180,E1 -6501.071,E2 -6501.071} C_VEL
LIN {X 0,Y 488.673,Z 193.617,A -85,B 0,C 180,E1 -6503.747,E2 -6503.747} C_VEL
LIN {X 0,Y 488.701,Z 193.606,A -85,B 0,C 180,E1 -6506.922,E2 -6506.922} C_VEL
LIN {X 0,Y 488.721,Z 193.605,A -85,B 0,C 180,E1 -6510.22,E2 -6510.22} C_VEL
LIN {X 0,Y 488.713,Z 193.611,A -85,B 0,C 180,E1 -6513.48,E2 -6513.48} C_VEL
LIN {X 0,Y 488.675,Z 193.609,A -85,B 0,C 180,E1 -6516.353,E2 -6516.353} C_VEL
LIN {X 0,Y 488.697,Z 193.612,A -85,B 0,C 180,E1 -6519.255,E2 -6519.255} C_VEL
LIN {X 0,Y 488.652,Z 193.612,A -85,B 0,C 180,E1 -6522.53,E2 -6522.53} C_VEL
LIN {X 0,Y 488.704,Z 193.612,A -85,B 0,C 180,E1 -6525.197,E2 -6525.197} C_VEL
LIN {X 0,Y 488.664,Z 193.611,A -85,B 0,C 180,E1 -6528.58,E2 -6528.58} C_VEL
LIN {X 0,Y 488.7,Z 193.611,A -85,B 0,C 180,E1 -6530.948,E2 -6530.948} C_VEL
LIN {X 0,Y 488.671,Z 193.61,A -85,B 0,C 180,E1 -6533.867,E2 -6533.867} C_VEL
LIN {X 0,Y 488.704,Z 193.612,A -85,B 0,C 180,E1 -6536.874,E2 -6536.874} C_VEL
LIN {X 0,Y 488.718,Z 193.605,A -85,B 0,C 180,E1 -6539.78,E2 -6539.78} C_VEL
LIN {X 0,Y 488.77,Z 193.705,A -85,B 0,C 180,E1 -6542.858,E2 -6542.858} C_VEL
LIN {X 0,Y 491.058,Z 205.528,A -85,B 0,C 180,E1 -6544.8,E2 -6544.8} C_VEL
LIN {X 0,Y 490.625,Z 220.232,A -85,B 0,C 180,E1 -6547.029,E2 -6547.029} C_VEL
LIN {X 0,Y 489.959,Z 240.677,A -85,B 0,C 180,E1 -6550.082,E2 -6550.082} C_VEL
LIN {X 0,Y 489.389,Z 259.626,A -85,B 0,C 180,E1 -6552.878,E2 -6552.878} C_VEL
LIN {X 0,Y 489.258,Z 265.674,A -85,B 0,C 180,E1 -6553.734,E2 -6553.734} C_VEL
LIN {X 0,Y 491.578,Z 283.878,A -85,B 0,C 180,E1 -6554.091,E2 -6554.091} C_VEL
LIN {X 0,Y 490.92,Z 375.094,A -85,B 0,C 180,E1 -6555.491,E2 -6555.491} C_VEL
LIN {X 0,Y 490.561,Z 388.876,A -85,B 0,C 180,E1 -6555.877,E2 -6555.877} C_VEL
LIN {X 0,Y 490.19,Z 401.822,A -85,B 0,C 180,E1 -6556.421,E2 -6556.421} C_VEL
LIN {X 0,Y 489.719,Z 413.309,A -85,B 0,C 180,E1 -6557.073,E2 -6557.073} C_VEL
LIN {X 0,Y 489.307,Z 424.485,A -85,B 0,C 180,E1 -6557.882,E2 -6557.882} C_VEL
LIN {X 0,Y 489.017,Z 434.821,A -85,B 0,C 180,E1 -6558.812,E2 -6558.812} C_VEL
LIN {X 0,Y 488.627,Z 444.188,A -85,B 0,C 180,E1 -6559.852,E2 -6559.852} C_VEL
LIN {X 0,Y 488.346,Z 453.285,A -85,B 0,C 180,E1 -6561.1,E2 -6561.1} C_VEL
LIN {X 0,Y 488.176,Z 460.617,A -85,B 0,C 180,E1 -6562.347,E2 -6562.347} C_VEL
LIN {X 0,Y 488.092,Z 465.985,A -85,B 0,C 180,E1 -6563.479,E2 -6563.479} C_VEL
LIN {X 0,Y 488.04,Z 470.378,A -85,B 0,C 180,E1 -6564.629,E2 -6564.629} C_VEL
LIN {X 0,Y 487.994,Z 474.049,A -85,B 0,C 180,E1 -6565.87,E2 -6565.87} C_VEL
LIN {X 0,Y 488.016,Z 475.944,A -85,B 0,C 180,E1 -6566.697,E2 -6566.697} C_VEL
LIN {X 0,Y 487.999,Z 477.361,A -85,B 0,C 180,E1 -6567.524,E2 -6567.524} C_VEL
LIN {X 0,Y 487.874,Z 478.963,A -85,B 0,C 180,E1 -6569.174,E2 -6569.174} C_VEL
LIN {X 0,Y 487.882,Z 479.171,A -85,B 0,C 180,E1 -6570,E2 -6570} C_VEL
LIN {X 0,Y 487.875,Z 478.935,A -85,B 0,C 180,E1 -6570.825,E2 -6570.825} C_VEL
LIN {X 0,Y 488.001,Z 477.274,A -85,B 0,C 180,E1 -6572.476,E2 -6572.476} C_VEL
LIN {X 0,Y 488.029,Z 475.831,A -85,B 0,C 180,E1 -6573.302,E2 -6573.302} C_VEL
LIN {X 0,Y 487.951,Z 472.798,A -85,B 0,C 180,E1 -6574.543,E2 -6574.543} C_VEL
LIN {X 0,Y 488.019,Z 468.712,A -85,B 0,C 180,E1 -6575.785,E2 -6575.785} C_VEL
LIN {X 0,Y 488.172,Z 462.432,A -85,B 0,C 180,E1 -6577.237,E2 -6577.237} C_VEL
LIN {X 0,Y 488.284,Z 455.576,A -85,B 0,C 180,E1 -6578.484,E2 -6578.484} C_VEL
LIN {X 0,Y 488.494,Z 447.08,A -85,B 0,C 180,E1 -6579.732,E2 -6579.732} C_VEL
LIN {X 0,Y 488.813,Z 438.349,A -85,B 0,C 180,E1 -6580.772,E2 -6580.772} C_VEL
LIN {X 0,Y 489.187,Z 427.853,A -85,B 0,C 180,E1 -6581.791,E2 -6581.791} C_VEL
LIN {X 0,Y 489.54,Z 417.246,A -85,B 0,C 180,E1 -6582.625,E2 -6582.625} C_VEL
LIN {X 0,Y 489.974,Z 405.2,A -85,B 0,C 180,E1 -6583.373,E2 -6583.373} C_VEL
LIN {X 0,Y 490.381,Z 393.02,A -85,B 0,C 180,E1 -6583.943,E2 -6583.943} C_VEL
LIN {X 0,Y 490.8,Z 379.84,A -85,B 0,C 180,E1 -6584.38,E2 -6584.38} C_VEL
LIN {X 0,Y 491.016,Z 367.243,A -85,B 0,C 180,E1 -6584.638,E2 -6584.638} C_VEL
LIN {X 0,Y 491.55,Z 282.67,A -85,B 0,C 180,E1 -6585.924,E2 -6585.924} C_VEL
LIN {X 0,Y 489.158,Z 264.156,A -85,B 0,C 180,E1 -6586.301,E2 -6586.301} C_VEL
LIN {X 0,Y 489.696,Z 241.935,A -85,B 0,C 180,E1 -6589.492,E2 -6589.492} C_VEL
LIN {X 0,Y 490.166,Z 222.347,A -85,B 0,C 180,E1 -6592.331,E2 -6592.331} C_VEL
LIN {X 0,Y 490.632,Z 204.144,A -85,B 0,C 180,E1 -6594.997,E2 -6594.997} C_VEL
LIN {X 0,Y 488.721,Z 193.611,A -85,B 0,C 180,E1 -6596.659,E2 -6596.659} C_VEL
LIN {X 0,Y 488.701,Z 193.615,A -85,B 0,C 180,E1 -6599.272,E2 -6599.272} C_VEL
LIN {X 0,Y 488.701,Z 193.609,A -85,B 0,C 180,E1 -6602.147,E2 -6602.147} C_VEL
LIN {X 0,Y 488.714,Z 193.61,A -85,B 0,C 180,E1 -6605.115,E2 -6605.115} C_VEL
LIN {X 0,Y 488.675,Z 193.612,A -85,B 0,C 180,E1 -6608.2,E2 -6608.2} C_VEL
LIN {X 0,Y 488.68,Z 193.61,A -85,B 0,C 180,E1 -6611.418,E2 -6611.418} C_VEL
LIN {X 0,Y 488.701,Z 193.61,A -85,B 0,C 180,E1 -6614.802,E2 -6614.802} C_VEL
LIN {X 0,Y 488.688,Z 193.606,A -85,B 0,C 180,E1 -6617.474,E2 -6617.474} C_VEL
LIN {X 0,Y 488.694,Z 193.612,A -85,B 0,C 180,E1 -6620.745,E2 -6620.745} C_VEL
LIN {X 0,Y 488.669,Z 193.613,A -85,B 0,C 180,E1 -6623.867,E2 -6623.867} C_VEL
LIN {X 0,Y 488.738,Z 193.602,A -85,B 0,C 180,E1 -6626.877,E2 -6626.877} C_VEL
LIN {X 0,Y 488.722,Z 193.607,A -85,B 0,C 180,E1 -6629.78,E2 -6629.78} C_VEL
LIN {X 0,Y 488.725,Z 193.602,A -85,B 0,C 180,E1 -6633.072,E2 -6633.072} C_VEL
LIN {X 0,Y 488.671,Z 193.614,A -85,B 0,C 180,E1 -6636.253,E2 -6636.253} C_VEL
LIN {X 0,Y 488.747,Z 193.6,A -85,B 0,C 180,E1 -6639.176,E2 -6639.176} C_VEL
LIN {X 0,Y 488.748,Z 193.606,A -85,B 0,C 180,E1 -6641.632,E2 -6641.632} C_VEL
LIN {X 0,Y 488.757,Z 193.599,A -85,B 0,C 180,E1 -6644.999,E2 -6644.999} C_VEL
LIN {X 0,Y 488.806,Z 193.592,A -85,B 0,C 180,E1 -6648.387,E2 -6648.387} C_VEL
LIN {X 0,Y 488.816,Z 193.599,A -85,B 0,C 180,E1 -6651.734,E2 -6651.734} C_VEL
LIN {X 0,Y 488.848,Z 193.589,A -85,B 0,C 180,E1 -6654.224,E2 -6654.224} C_VEL
LIN {X 0,Y 488.961,Z 193.58,A -85,B 0,C 180,E1 -6657.529,E2 -6657.529} C_VEL
LIN {X 0,Y 488.934,Z 193.58,A -85,B 0,C 180,E1 -6660.824,E2 -6660.824} C_VEL
LIN {X 0,Y 488.961,Z 193.575,A -85,B 0,C 180,E1 -6662.471,E2 -6662.471} C_VEL
LIN {X 0,Y 488.842,Z 193.591,A -85,B 0,C 180,E1 -6665.776,E2 -6665.776} C_VEL
LIN {X 0,Y 488.785,Z 193.597,A -85,B 0,C 180,E1 -6668.267,E2 -6668.267} C_VEL
LIN {X 0,Y 488.806,Z 193.598,A -85,B 0,C 180,E1 -6671.612,E2 -6671.612} C_VEL
LIN {X 0,Y 488.762,Z 193.608,A -85,B 0,C 180,E1 -6675,E2 -6675} C_VEL
LIN {X 0,Y 488.747,Z 193.606,A -85,B 0,C 180,E1 -6678.442,E2 -6678.442} C_VEL
LIN {X 0,Y 488.784,Z 193.742,A -85,B 0,C 180,E1 -6681.021,E2 -6681.021} C_VEL
LIN {X 0,Y 489.439,Z 197.747,A -85,B 0,C 180,E1 -6681.783,E2 -6681.783} C_VEL
LIN {X 0,Y 491.929,Z 209.108,A -85,B 0,C 180,E1 -6682.053,E2 -6682.053} C_VEL
LIN {X 0,Y 491.129,Z 305.289,A -85,B 0,C 180,E1 -6683.549,E2 -6683.549} C_VEL
LIN {X 0,Y 490.952,Z 318.705,A -85,B 0,C 180,E1 -6683.932,E2 -6683.932} C_VEL
LIN {X 0,Y 490.667,Z 331.644,A -85,B 0,C 180,E1 -6684.481,E2 -6684.481} C_VEL
LIN {X 0,Y 490.375,Z 342.825,A -85,B 0,C 180,E1 -6685.124,E2 -6685.124} C_VEL
LIN {X 0,Y 489.975,Z 354.02,A -85,B 0,C 180,E1 -6685.943,E2 -6685.943} C_VEL
LIN {X 0,Y 489.627,Z 363.768,A -85,B 0,C 180,E1 -6686.831,E2 -6686.831} C_VEL
LIN {X 0,Y 489.284,Z 372.734,A -85,B 0,C 180,E1 -6687.828,E2 -6687.828} C_VEL
LIN {X 0,Y 488.94,Z 381.049,A -85,B 0,C 180,E1 -6688.967,E2 -6688.967} C_VEL
LIN {X 0,Y 488.627,Z 389.128,A -85,B 0,C 180,E1 -6690.346,E2 -6690.346} C_VEL
LIN {X 0,Y 488.442,Z 394.681,A -85,B 0,C 180,E1 -6691.543,E2 -6691.543} C_VEL
LIN {X 0,Y 488.251,Z 398.86,A -85,B 0,C 180,E1 -6692.669,E2 -6692.669} C_VEL
LIN {X 0,Y 488.133,Z 403.04,A -85,B 0,C 180,E1 -6694.16,E2 -6694.16} C_VEL
LIN {X 0,Y 488.026,Z 405.024,A -85,B 0,C 180,E1 -6695.172,E2 -6695.172} C_VEL
LIN {X 0,Y 487.979,Z 406.468,A -85,B 0,C 180,E1 -6696.242,E2 -6696.242} C_VEL
LIN {X 0,Y 487.93,Z 407.323,A -85,B 0,C 180,E1 -6697.608,E2 -6697.608} C_VEL
LIN {X 0,Y 487.941,Z 406.88,A -85,B 0,C 180,E1 -6699.327,E2 -6699.327} C_VEL
LIN {X 0,Y 487.975,Z 405.698,A -85,B 0,C 180,E1 -6700.399,E2 -6700.399} C_VEL
LIN {X 0,Y 488.131,Z 402.63,A -85,B 0,C 180,E1 -6702.028,E2 -6702.028} C_VEL
LIN {X 0,Y 488.236,Z 399.372,A -85,B 0,C 180,E1 -6703.196,E2 -6703.196} C_VEL
LIN {X 0,Y 488.366,Z 394.777,A -85,B 0,C 180,E1 -6704.452,E2 -6704.452} C_VEL
LIN {X 0,Y 488.557,Z 388.658,A -85,B 0,C 180,E1 -6705.768,E2 -6705.768} C_VEL
LIN {X 0,Y 488.888,Z 380.454,A -85,B 0,C 180,E1 -6707.151,E2 -6707.151} C_VEL
LIN {X 0,Y 488.982,Z 378.214,A -85,B 0,C 180,E1 -6707.475,E2 -6707.475} C_VEL
LIN {X 0,Y 488.492,Z 374.455,A -85,B 0,C 180,E1 -6708.002,E2 -6708.002} C_VEL
LIN {X 0,Y 485.985,Z 368.091,A -85,B 0,C 180,E1 -6708.845,E2 -6708.845} C_VEL
LIN {X 0,Y 483.437,Z 361.231,A -85,B 0,C 180,E1 -6709.636,E2 -6709.636} C_VEL
LIN {X 0,Y 482.888,Z 356.639,A -85,B 0,C 180,E1 -6710.079,E2 -6710.079} C_VEL
LIN {X 0,Y 483.265,Z 345.402,A -85,B 0,C 180,E1 -6710.959,E2 -6710.959} C_VEL
LIN {X 0,Y 483.699,Z 333.434,A -85,B 0,C 180,E1 -6711.684,E2 -6711.684} C_VEL
LIN {X 0,Y 483.985,Z 321.538,A -85,B 0,C 180,E1 -6712.232,E2 -6712.232} C_VEL
LIN {X 0,Y 484.18,Z 309.012,A -85,B 0,C 180,E1 -6712.64,E2 -6712.64} C_VEL
LIN {X 0,Y 484.345,Z 294.913,A -85,B 0,C 180,E1 -6712.911,E2 -6712.911} C_VEL
LIN {X 0,Y 484.849,Z 208.846,A -85,B 0,C 180,E1 -6714.244,E2 -6714.244} C_VEL
LIN {X 0,Y 482.277,Z 197.707,A -85,B 0,C 180,E1 -6714.51,E2 -6714.51} C_VEL
LIN {X 0,Y 481.723,Z 194.483,A -85,B 0,C 180,E1 -6715.204,E2 -6715.204} C_VEL
LIN {X 0,Y 481.644,Z 194.487,A -85,B 0,C 180,E1 -6718.312,E2 -6718.312} C_VEL
LIN {X 0,Y 481.698,Z 194.486,A -85,B 0,C 180,E1 -6721.219,E2 -6721.219} C_VEL
LIN {X 0,Y 481.671,Z 194.481,A -85,B 0,C 180,E1 -6724.041,E2 -6724.041} C_VEL
LIN {X 0,Y 481.675,Z 194.486,A -85,B 0,C 180,E1 -6726.812,E2 -6726.812} C_VEL
LIN {X 0,Y 481.695,Z 194.48,A -85,B 0,C 180,E1 -6729.503,E2 -6729.503} C_VEL
LIN {X 0,Y 481.689,Z 194.479,A -85,B 0,C 180,E1 -6732.158,E2 -6732.158} C_VEL
LIN {X 0,Y 481.743,Z 194.48,A -85,B 0,C 180,E1 -6734.776,E2 -6734.776} C_VEL
LIN {X 0,Y 481.752,Z 194.473,A -85,B 0,C 180,E1 -6738.215,E2 -6738.215} C_VEL
LIN {X 0,Y 481.741,Z 194.473,A -85,B 0,C 180,E1 -6741.612,E2 -6741.612} C_VEL
LIN {X 0,Y 481.801,Z 194.467,A -85,B 0,C 180,E1 -6744.14,E2 -6744.14} C_VEL
LIN {X 0,Y 481.922,Z 194.45,A -85,B 0,C 180,E1 -6747.493,E2 -6747.493} C_VEL
LIN {X 0,Y 481.941,Z 194.45,A -85,B 0,C 180,E1 -6750,E2 -6750} C_VEL
LIN {X 0,Y 481.919,Z 194.458,A -85,B 0,C 180,E1 -6752.508,E2 -6752.508} C_VEL
LIN {X 0,Y 481.799,Z 194.467,A -85,B 0,C 180,E1 -6755.861,E2 -6755.861} C_VEL
LIN {X 0,Y 481.742,Z 194.48,A -85,B 0,C 180,E1 -6758.389,E2 -6758.389} C_VEL
LIN {X 0,Y 481.753,Z 194.474,A -85,B 0,C 180,E1 -6761.785,E2 -6761.785} C_VEL
LIN {X 0,Y 481.742,Z 194.473,A -85,B 0,C 180,E1 -6765.224,E2 -6765.224} C_VEL
LIN {X 0,Y 481.709,Z 194.477,A -85,B 0,C 180,E1 -6768.722,E2 -6768.722} C_VEL
LIN {X 0,Y 481.647,Z 194.486,A -85,B 0,C 180,E1 -6771.395,E2 -6771.395} C_VEL
LIN {X 0,Y 481.651,Z 194.49,A -85,B 0,C 180,E1 -6774.115,E2 -6774.115} C_VEL
LIN {X 0,Y 481.695,Z 194.479,A -85,B 0,C 180,E1 -6777.127,E2 -6777.127} C_VEL
LIN {X 0,Y 481.674,Z 194.489,A -85,B 0,C 180,E1 -6779.742,E2 -6779.742} C_VEL
LIN {X 0,Y 481.674,Z 194.481,A -85,B 0,C 180,E1 -6782.674,E2 -6782.674} C_VEL
LIN {X 0,Y 481.663,Z 194.485,A -85,B 0,C 180,E1 -6785.204,E2 -6785.204} C_VEL
LIN {X 0,Y 481.668,Z 194.482,A -85,B 0,C 180,E1 -6788.86,E2 -6788.86} C_VEL
LIN {X 0,Y 481.642,Z 194.486,A -85,B 0,C 180,E1 -6792.162,E2 -6792.162} C_VEL
LIN {X 0,Y 481.656,Z 194.49,A -85,B 0,C 180,E1 -6795.542,E2 -6795.542} C_VEL
LIN {X 0,Y 481.635,Z 194.489,A -85,B 0,C 180,E1 -6798.956,E2 -6798.956} C_VEL
LIN {X 0,Y 481.654,Z 194.484,A -85,B 0,C 180,E1 -6801.993,E2 -6801.993} C_VEL
LIN {X 0,Y 481.686,Z 194.486,A -85,B 0,C 180,E1 -6805.318,E2 -6805.318} C_VEL
LIN {X 0,Y 481.646,Z 194.485,A -85,B 0,C 180,E1 -6808.312,E2 -6808.312} C_VEL
LIN {X 0,Y 481.663,Z 194.488,A -85,B 0,C 180,E1 -6811.216,E2 -6811.216} C_VEL
LIN {X 0,Y 481.667,Z 194.482,A -85,B 0,C 180,E1 -6814.041,E2 -6814.041} C_VEL
LIN {X 0,Y 481.677,Z 194.488,A -85,B 0,C 180,E1 -6816.812,E2 -6816.812} C_VEL
LIN {X 0,Y 481.698,Z 194.479,A -85,B 0,C 180,E1 -6819.503,E2 -6819.503} C_VEL
LIN {X 0,Y 481.69,Z 194.48,A -85,B 0,C 180,E1 -6822.158,E2 -6822.158} C_VEL
LIN {X 0,Y 481.741,Z 194.48,A -85,B 0,C 180,E1 -6824.776,E2 -6824.776} C_VEL
LIN {X 0,Y 481.754,Z 194.474,A -85,B 0,C 180,E1 -6828.215,E2 -6828.215} C_VEL
LIN {X 0,Y 481.739,Z 194.473,A -85,B 0,C 180,E1 -6831.611,E2 -6831.611} C_VEL
LIN {X 0,Y 481.791,Z 194.47,A -85,B 0,C 180,E1 -6834.139,E2 -6834.139} C_VEL
LIN {X 0,Y 481.921,Z 194.45,A -85,B 0,C 180,E1 -6837.493,E2 -6837.493} C_VEL
LIN {X 0,Y 481.917,Z 194.454,A -85,B 0,C 180,E1 -6840,E2 -6840} C_VEL
LIN {X 0,Y 481.912,Z 194.457,A -85,B 0,C 180,E1 -6842.508,E2 -6842.508} C_VEL
LIN {X 0,Y 481.779,Z 194.471,A -85,B 0,C 180,E1 -6845.861,E2 -6845.861} C_VEL
LIN {X 0,Y 481.724,Z 194.48,A -85,B 0,C 180,E1 -6848.389,E2 -6848.389} C_VEL
LIN {X 0,Y 481.754,Z 194.475,A -85,B 0,C 180,E1 -6851.785,E2 -6851.785} C_VEL
LIN {X 0,Y 481.733,Z 194.474,A -85,B 0,C 180,E1 -6855.225,E2 -6855.225} C_VEL
LIN {X 0,Y 481.708,Z 194.477,A -85,B 0,C 180,E1 -6858.722,E2 -6858.722} C_VEL
LIN {X 0,Y 481.648,Z 194.487,A -85,B 0,C 180,E1 -6861.395,E2 -6861.395} C_VEL
LIN {X 0,Y 481.651,Z 194.488,A -85,B 0,C 180,E1 -6864.115,E2 -6864.115} C_VEL
LIN {X 0,Y 481.656,Z 194.485,A -85,B 0,C 180,E1 -6867.117,E2 -6867.117} C_VEL
LIN {X 0,Y 481.669,Z 194.489,A -85,B 0,C 180,E1 -6869.742,E2 -6869.742} C_VEL
LIN {X 0,Y 481.655,Z 194.483,A -85,B 0,C 180,E1 -6872.676,E2 -6872.676} C_VEL
LIN {X 0,Y 481.633,Z 194.492,A -85,B 0,C 180,E1 -6875.71,E2 -6875.71} C_VEL
LIN {X 0,Y 481.669,Z 194.483,A -85,B 0,C 180,E1 -6878.859,E2 -6878.859} C_VEL
LIN {X 0,Y 481.618,Z 194.488,A -85,B 0,C 180,E1 -6882.164,E2 -6882.164} C_VEL
LIN {X 0,Y 481.656,Z 194.483,A -85,B 0,C 180,E1 -6884.458,E2 -6884.458} C_VEL
LIN {X 0,Y 481.618,Z 194.491,A -85,B 0,C 180,E1 -6886.855,E2 -6886.855} C_VEL
LIN {X 0,Y 481.659,Z 194.483,A -85,B 0,C 180,E1 -6890.057,E2 -6890.057} C_VEL
LIN {X 0,Y 481.622,Z 194.494,A -85,B 0,C 180,E1 -6893.252,E2 -6893.252} C_VEL
LIN {X 0,Y 481.673,Z 194.482,A -85,B 0,C 180,E1 -6896.327,E2 -6896.327} C_VEL
LIN {X 0,Y 481.645,Z 194.489,A -85,B 0,C 180,E1 -6899.419,E2 -6899.419} C_VEL
LIN {X 0,Y 481.692,Z 194.585,A -85,B 0,C 180,E1 -6902.652,E2 -6902.652} C_VEL
LIN {X 0,Y 484.101,Z 206.593,A -85,B 0,C 180,E1 -6904.66,E2 -6904.66} C_VEL
LIN {X 0,Y 483.696,Z 221.156,A -85,B 0,C 180,E1 -6906.902,E2 -6906.902} C_VEL
LIN {X 0,Y 482.968,Z 241.621,A -85,B 0,C 180,E1 -6910.003,E2 -6910.003} C_VEL
LIN {X 0,Y 482.29,Z 263.338,A -85,B 0,C 180,E1 -6913.252,E2 -6913.252} C_VEL
LIN {X 0,Y 482.268,Z 265.042,A -85,B 0,C 180,E1 -6913.496,E2 -6913.496} C_VEL
LIN {X 0,Y 484.739,Z 284.881,A -85,B 0,C 180,E1 -6913.891,E2 -6913.891} C_VEL
LIN {X 0,Y 484.048,Z 374.131,A -85,B 0,C 180,E1 -6915.28,E2 -6915.28} C_VEL
LIN {X 0,Y 483.681,Z 387.302,A -85,B 0,C 180,E1 -6915.645,E2 -6915.645} C_VEL
LIN {X 0,Y 483.302,Z 400.031,A -85,B 0,C 180,E1 -6916.171,E2 -6916.171} C_VEL
LIN {X 0,Y 482.783,Z 412.173,A -85,B 0,C 180,E1 -6916.852,E2 -6916.852} C_VEL
LIN {X 0,Y 482.327,Z 423.184,A -85,B 0,C 180,E1 -6917.649,E2 -6917.649} C_VEL
LIN {X 0,Y 482.041,Z 433.143,A -85,B 0,C 180,E1 -6918.542,E2 -6918.542} C_VEL
LIN {X 0,Y 481.658,Z 441.873,A -85,B 0,C 180,E1 -6919.491,E2 -6919.491} C_VEL
LIN {X 0,Y 481.391,Z 449.925,A -85,B 0,C 180,E1 -6920.546,E2 -6920.546} C_VEL
LIN {X 0,Y 481.156,Z 457.804,A -85,B 0,C 180,E1 -6921.812,E2 -6921.812} C_VEL
LIN {X 0,Y 480.975,Z 465.028,A -85,B 0,C 180,E1 -6923.287,E2 -6923.287} C_VEL
LIN {X 0,Y 480.946,Z 469.846,A -85,B 0,C 180,E1 -6924.549,E2 -6924.549} C_VEL
LIN {X 0,Y 480.891,Z 473.522,A -85,B 0,C 180,E1 -6925.809,E2 -6925.809} C_VEL
LIN {X 0,Y 480.938,Z 475.421,A -85,B 0,C 180,E1 -6926.649,E2 -6926.649} C_VEL
LIN {X 0,Y 480.937,Z 476.842,A -85,B 0,C 180,E1 -6927.487,E2 -6927.487} C_VEL
LIN {X 0,Y 480.797,Z 478.443,A -85,B 0,C 180,E1 -6929.162,E2 -6929.162} C_VEL
LIN {X 0,Y 480.802,Z 478.651,A -85,B 0,C 180,E1 -6930,E2 -6930} C_VEL
LIN {X 0,Y 480.798,Z 478.414,A -85,B 0,C 180,E1 -6930.837,E2 -6930.837} C_VEL
LIN {X 0,Y 480.94,Z 476.747,A -85,B 0,C 180,E1 -6932.512,E2 -6932.512} C_VEL
LIN {X 0,Y 480.952,Z 475.298,A -85,B 0,C 180,E1 -6933.351,E2 -6933.351} C_VEL
LIN {X 0,Y 480.864,Z 472.257,A -85,B 0,C 180,E1 -6934.61,E2 -6934.61} C_VEL
LIN {X 0,Y 480.923,Z 468.161,A -85,B 0,C 180,E1 -6935.871,E2 -6935.871} C_VEL
LIN {X 0,Y 481.095,Z 461.871,A -85,B 0,C 180,E1 -6937.344,E2 -6937.344} C_VEL
LIN {X 0,Y 481.206,Z 455.007,A -85,B 0,C 180,E1 -6938.609,E2 -6938.609} C_VEL
LIN {X 0,Y 481.43,Z 446.502,A -85,B 0,C 180,E1 -6939.876,E2 -6939.876} C_VEL
LIN {X 0,Y 481.797,Z 437.765,A -85,B 0,C 180,E1 -6940.931,E2 -6940.931} C_VEL
LIN {X 0,Y 482.163,Z 427.524,A -85,B 0,C 180,E1 -6941.941,E2 -6941.941} C_VEL
LIN {X 0,Y 482.598,Z 416.344,A -85,B 0,C 180,E1 -6942.831,E2 -6942.831} C_VEL
LIN {X 0,Y 483.054,Z 404.571,A -85,B 0,C 180,E1 -6943.568,E2 -6943.568} C_VEL
LIN {X 0,Y 483.469,Z 392.383,A -85,B 0,C 180,E1 -6944.146,E2 -6944.146} C_VEL
LIN {X 0,Y 483.893,Z 379.197,A -85,B 0,C 180,E1 -6944.59,E2 -6944.59} C_VEL
LIN {X 0,Y 484.141,Z 366.585,A -85,B 0,C 180,E1 -6944.851,E2 -6944.851} C_VEL
LIN {X 0,Y 484.621,Z 282.944,A -85,B 0,C 180,E1 -6946.15,E2 -6946.15} C_VEL
LIN {X 0,Y 482.151,Z 263.447,A -85,B 0,C 180,E1 -6946.568,E2 -6946.568} C_VEL
LIN {X 0,Y 482.756,Z 241.366,A -85,B 0,C 180,E1 -6949.784,E2 -6949.784} C_VEL
LIN {X 0,Y 483.257,Z 221.787,A -85,B 0,C 180,E1 -6952.668,E2 -6952.668} C_VEL
LIN {X 0,Y 483.69,Z 205.38,A -85,B 0,C 180,E1 -6955.107,E2 -6955.107} C_VEL
LIN {X 0,Y 481.678,Z 194.488,A -85,B 0,C 180,E1 -6956.863,E2 -6956.863} C_VEL
LIN {X 0,Y 481.666,Z 194.489,A -85,B 0,C 180,E1 -6959.742,E2 -6959.742} C_VEL
LIN {X 0,Y 481.67,Z 194.489,A -85,B 0,C 180,E1 -6962.674,E2 -6962.674} C_VEL
LIN {X 0,Y 481.632,Z 194.488,A -85,B 0,C 180,E1 -6965.71,E2 -6965.71} C_VEL
LIN {X 0,Y 481.666,Z 194.488,A -85,B 0,C 180,E1 -6968.859,E2 -6968.859} C_VEL
LIN {X 0,Y 481.64,Z 194.488,A -85,B 0,C 180,E1 -6972.161,E2 -6972.161} C_VEL
LIN {X 0,Y 481.654,Z 194.483,A -85,B 0,C 180,E1 -6975.542,E2 -6975.542} C_VEL
LIN {X 0,Y 481.634,Z 194.488,A -85,B 0,C 180,E1 -6978.956,E2 -6978.956} C_VEL
LIN {X 0,Y 481.649,Z 194.488,A -85,B 0,C 180,E1 -6981.993,E2 -6981.993} C_VEL
LIN {X 0,Y 481.688,Z 194.479,A -85,B 0,C 180,E1 -6985.318,E2 -6985.318} C_VEL
LIN {X 0,Y 481.645,Z 194.491,A -85,B 0,C 180,E1 -6988.311,E2 -6988.311} C_VEL
LIN {X 0,Y 481.674,Z 194.481,A -85,B 0,C 180,E1 -6991.217,E2 -6991.217} C_VEL
LIN {X 0,Y 481.664,Z 194.488,A -85,B 0,C 180,E1 -6994.041,E2 -6994.041} C_VEL
LIN {X 0,Y 481.674,Z 194.481,A -85,B 0,C 180,E1 -6996.812,E2 -6996.812} C_VEL
LIN {X 0,Y 481.695,Z 194.481,A -85,B 0,C 180,E1 -6999.503,E2 -6999.503} C_VEL
LIN {X 0,Y 481.687,Z 194.482,A -85,B 0,C 180,E1 -7002.158,E2 -7002.158} C_VEL
LIN {X 0,Y 481.74,Z 194.473,A -85,B 0,C 180,E1 -7004.776,E2 -7004.776} C_VEL
LIN {X 0,Y 481.751,Z 194.472,A -85,B 0,C 180,E1 -7008.215,E2 -7008.215} C_VEL
LIN {X 0,Y 481.762,Z 194.476,A -85,B 0,C 180,E1 -7011.612,E2 -7011.612} C_VEL
LIN {X 0,Y 481.808,Z 194.466,A -85,B 0,C 180,E1 -7014.139,E2 -7014.139} C_VEL
LIN {X 0,Y 481.928,Z 194.457,A -85,B 0,C 180,E1 -7017.492,E2 -7017.492} C_VEL
LIN {X 0,Y 481.886,Z 194.458,A -85,B 0,C 180,E1 -7020.836,E2 -7020.836} C_VEL
LIN {X 0,Y 481.928,Z 194.452,A -85,B 0,C 180,E1 -7022.507,E2 -7022.507} C_VEL
LIN {X 0,Y 481.801,Z 194.467,A -85,B 0,C 180,E1 -7025.861,E2 -7025.861} C_VEL
LIN {X 0,Y 481.74,Z 194.475,A -85,B 0,C 180,E1 -7028.389,E2 -7028.389} C_VEL
LIN {X 0,Y 481.751,Z 194.476,A -85,B 0,C 180,E1 -7031.785,E2 -7031.785} C_VEL
LIN {X 0,Y 481.743,Z 194.481,A -85,B 0,C 180,E1 -7035.224,E2 -7035.224} C_VEL
LIN {X 0,Y 481.71,Z 194.484,A -85,B 0,C 180,E1 -7038.722,E2 -7038.722} C_VEL
LIN {X 0,Y 481.768,Z 194.588,A -85,B 0,C 180,E1 -7040.828,E2 -7040.828} C_VEL
LIN {X 0,Y 482.454,Z 198.367,A -85,B 0,C 180,E1 -7041.532,E2 -7041.532} C_VEL
LIN {X 0,Y 485.122,Z 209.724,A -85,B 0,C 180,E1 -7041.818,E2 -7041.818} C_VEL
LIN {X 0,Y 484.298,Z 305.327,A -85,B 0,C 180,E1 -7043.328,E2 -7043.328} C_VEL
LIN {X 0,Y 484.093,Z 318.815,A -85,B 0,C 180,E1 -7043.713,E2 -7043.713} C_VEL
LIN {X 0,Y 483.834,Z 331.004,A -85,B 0,C 180,E1 -7044.227,E2 -7044.227} C_VEL
LIN {X 0,Y 483.485,Z 343.295,A -85,B 0,C 180,E1 -7044.932,E2 -7044.932} C_VEL
LIN {X 0,Y 483.051,Z 354.65,A -85,B 0,C 180,E1 -7045.775,E2 -7045.775} C_VEL
LIN {X 0,Y 482.688,Z 364.766,A -85,B 0,C 180,E1 -7046.714,E2 -7046.714} C_VEL
LIN {X 0,Y 482.287,Z 374.158,A -85,B 0,C 180,E1 -7047.795,E2 -7047.795} C_VEL
LIN {X 0,Y 481.879,Z 383.198,A -85,B 0,C 180,E1 -7049.088,E2 -7049.088} C_VEL
LIN {X 0,Y 481.594,Z 390.263,A -85,B 0,C 180,E1 -7050.35,E2 -7050.35} C_VEL
LIN {X 0,Y 481.352,Z 396.257,A -85,B 0,C 180,E1 -7051.71,E2 -7051.71} C_VEL
LIN {X 0,Y 481.136,Z 401.164,A -85,B 0,C 180,E1 -7053.17,E2 -7053.17} C_VEL
LIN {X 0,Y 480.983,Z 404.896,A -85,B 0,C 180,E1 -7054.74,E2 -7054.74} C_VEL
LIN {X 0,Y 480.926,Z 406.486,A -85,B 0,C 180,E1 -7055.77,E2 -7055.77} C_VEL
LIN {X 0,Y 480.868,Z 407.508,A -85,B 0,C 180,E1 -7056.814,E2 -7056.814} C_VEL
LIN {X 0,Y 480.843,Z 407.893,A -85,B 0,C 180,E1 -7057.883,E2 -7057.883} C_VEL
LIN {X 0,Y 480.87,Z 407.465,A -85,B 0,C 180,E1 -7059.231,E2 -7059.231} C_VEL
LIN {X 0,Y 480.914,Z 406.057,A -85,B 0,C 180,E1 -7060.543,E2 -7060.543} C_VEL
LIN {X 0,Y 481.069,Z 402.777,A -85,B 0,C 180,E1 -7062.223,E2 -7062.223} C_VEL
LIN {X 0,Y 481.179,Z 399.605,A -85,B 0,C 180,E1 -7063.352,E2 -7063.352} C_VEL
LIN {X 0,Y 481.38,Z 394.402,A -85,B 0,C 180,E1 -7064.75,E2 -7064.75} C_VEL
LIN {X 0,Y 481.599,Z 387.48,A -85,B 0,C 180,E1 -7066.188,E2 -7066.188} C_VEL
LIN {X 0,Y 481.906,Z 380.399,A -85,B 0,C 180,E1 -7067.36,E2 -7067.36} C_VEL
LIN {X 0,Y 482.28,Z 372.185,A -85,B 0,C 180,E1 -7068.468,E2 -7068.468} C_VEL
LIN {X 0,Y 482.633,Z 362.667,A -85,B 0,C 180,E1 -7069.516,E2 -7069.516} C_VEL
LIN {X 0,Y 482.888,Z 356.639,A -85,B 0,C 180,E1 -7070.079,E2 -7070.079} C_VEL
LIN {X 0,Y 482.351,Z 351.926,A -85,B 0,C 180,E1 -7070.5,E2 -7070.5} C_VEL
LIN {X 0,Y 479.858,Z 344.1,A -85,B 0,C 180,E1 -7071.165,E2 -7071.165} C_VEL
LIN {X 0,Y 477.394,Z 335.872,A -85,B 0,C 180,E1 -7071.752,E2 -7071.752} C_VEL
LIN {X 0,Y 476.892,Z 330.539,A -85,B 0,C 180,E1 -7072.047,E2 -7072.047} C_VEL
LIN {X 0,Y 477.119,Z 317.572,A -85,B 0,C 180,E1 -7072.593,E2 -7072.593} C_VEL
LIN {X 0,Y 477.35,Z 304.658,A -85,B 0,C 180,E1 -7072.956,E2 -7072.956} C_VEL
LIN {X 0,Y 478.064,Z 209.89,A -85,B 0,C 180,E1 -7074.464,E2 -7074.464} C_VEL
LIN {X 0,Y 475.456,Z 199.164,A -85,B 0,C 180,E1 -7074.73,E2 -7074.73} C_VEL
LIN {X 0,Y 475.147,Z 197.959,A -85,B 0,C 180,E1 -7074.77,E2 -7074.77} C_VEL
LIN {X 0,Y 474.683,Z 195.36,A -85,B 0,C 180,E1 -7075.378,E2 -7075.378} C_VEL
LIN {X 0,Y 474.598,Z 195.368,A -85,B 0,C 180,E1 -7078.783,E2 -7078.783} C_VEL
LIN {X 0,Y 474.64,Z 195.359,A -85,B 0,C 180,E1 -7081.717,E2 -7081.717} C_VEL
LIN {X 0,Y 474.628,Z 195.361,A -85,B 0,C 180,E1 -7084.589,E2 -7084.589} C_VEL
LIN {X 0,Y 474.6,Z 195.366,A -85,B 0,C 180,E1 -7087.356,E2 -7087.356} C_VEL
LIN {X 0,Y 474.653,Z 195.356,A -85,B 0,C 180,E1 -7090.09,E2 -7090.09} C_VEL
LIN {X 0,Y 474.635,Z 195.364,A -85,B 0,C 180,E1 -7092.774,E2 -7092.774} C_VEL
LIN {X 0,Y 474.645,Z 195.358,A -85,B 0,C 180,E1 -7095.421,E2 -7095.421} C_VEL
LIN {X 0,Y 474.706,Z 195.349,A -85,B 0,C 180,E1 -7098.038,E2 -7098.038} C_VEL
LIN {X 0,Y 474.712,Z 195.349,A -85,B 0,C 180,E1 -7101.486,E2 -7101.486} C_VEL
LIN {X 0,Y 474.747,Z 195.348,A -85,B 0,C 180,E1 -7104.904,E2 -7104.904} C_VEL
LIN {X 0,Y 474.888,Z 195.326,A -85,B 0,C 180,E1 -7107.456,E2 -7107.456} C_VEL
LIN {X 0,Y 474.911,Z 195.325,A -85,B 0,C 180,E1 -7110,E2 -7110} C_VEL
LIN {X 0,Y 474.884,Z 195.334,A -85,B 0,C 180,E1 -7112.545,E2 -7112.545} C_VEL
LIN {X 0,Y 474.76,Z 195.345,A -85,B 0,C 180,E1 -7115.948,E2 -7115.948} C_VEL
LIN {X 0,Y 474.714,Z 195.353,A -85,B 0,C 180,E1 -7118.514,E2 -7118.514} C_VEL
LIN {X 0,Y 474.706,Z 195.354,A -85,B 0,C 180,E1 -7121.963,E2 -7121.963} C_VEL
LIN {X 0,Y 474.7,Z 195.351,A -85,B 0,C 180,E1 -7125.456,E2 -7125.456} C_VEL
LIN {X 0,Y 474.663,Z 195.354,A -85,B 0,C 180,E1 -7129.011,E2 -7129.011} C_VEL
LIN {X 0,Y 474.59,Z 195.368,A -85,B 0,C 180,E1 -7131.729,E2 -7131.729} C_VEL
LIN {X 0,Y 474.629,Z 195.36,A -85,B 0,C 180,E1 -7134.495,E2 -7134.495} C_VEL
LIN {X 0,Y 474.639,Z 195.359,A -85,B 0,C 180,E1 -7137.324,E2 -7137.324} C_VEL
LIN {X 0,Y 474.603,Z 195.364,A -85,B 0,C 180,E1 -7140.231,E2 -7140.231} C_VEL
LIN {X 0,Y 474.645,Z 195.359,A -85,B 0,C 180,E1 -7143.22,E2 -7143.22} C_VEL
LIN {X 0,Y 474.586,Z 195.365,A -85,B 0,C 180,E1 -7146.324,E2 -7146.324} C_VEL
LIN {X 0,Y 474.624,Z 195.367,A -85,B 0,C 180,E1 -7149.548,E2 -7149.548} C_VEL
LIN {X 0,Y 474.6,Z 195.363,A -85,B 0,C 180,E1 -7152.233,E2 -7152.233} C_VEL
LIN {X 0,Y 474.618,Z 195.366,A -85,B 0,C 180,E1 -7155.298,E2 -7155.298} C_VEL
LIN {X 0,Y 474.611,Z 195.361,A -85,B 0,C 180,E1 -7158.213,E2 -7158.213} C_VEL
LIN {X 0,Y 474.611,Z 195.365,A -85,B 0,C 180,E1 -7161.543,E2 -7161.543} C_VEL
LIN {X 0,Y 474.623,Z 195.362,A -85,B 0,C 180,E1 -7164.726,E2 -7164.726} C_VEL
LIN {X 0,Y 474.637,Z 195.359,A -85,B 0,C 180,E1 -7167.788,E2 -7167.788} C_VEL
LIN {X 0,Y 474.602,Z 195.368,A -85,B 0,C 180,E1 -7170.89,E2 -7170.89} C_VEL
LIN {X 0,Y 474.615,Z 195.361,A -85,B 0,C 180,E1 -7173.626,E2 -7173.626} C_VEL
LIN {X 0,Y 474.637,Z 195.362,A -85,B 0,C 180,E1 -7176.642,E2 -7176.642} C_VEL
LIN {X 0,Y 474.655,Z 195.356,A -85,B 0,C 180,E1 -7180.09,E2 -7180.09} C_VEL
LIN {X 0,Y 474.635,Z 195.366,A -85,B 0,C 180,E1 -7182.774,E2 -7182.774} C_VEL
LIN {X 0,Y 474.64,Z 195.358,A -85,B 0,C 180,E1 -7185.421,E2 -7185.421} C_VEL
LIN {X 0,Y 474.708,Z 195.35,A -85,B 0,C 180,E1 -7188.038,E2 -7188.038} C_VEL
LIN {X 0,Y 474.711,Z 195.348,A -85,B 0,C 180,E1 -7191.486,E2 -7191.486} C_VEL
LIN {X 0,Y 474.752,Z 195.346,A -85,B 0,C 180,E1 -7194.052,E2 -7194.052} C_VEL
LIN {X 0,Y 474.887,Z 195.326,A -85,B 0,C 180,E1 -7197.455,E2 -7197.455} C_VEL
LIN {X 0,Y 474.886,Z 195.33,A -85,B 0,C 180,E1 -7200,E2 -7200} C_VEL
LIN {X 0,Y 474.877,Z 195.333,A -85,B 0,C 180,E1 -7202.545,E2 -7202.545} C_VEL
LIN {X 0,Y 474.742,Z 195.349,A -85,B 0,C 180,E1 -7205.948,E2 -7205.948} C_VEL
LIN {X 0,Y 474.699,Z 195.353,A -85,B 0,C 180,E1 -7208.514,E2 -7208.514} C_VEL
LIN {X 0,Y 474.708,Z 195.355,A -85,B 0,C 180,E1 -7211.962,E2 -7211.962} C_VEL
LIN {X 0,Y 474.691,Z 195.353,A -85,B 0,C 180,E1 -7215.456,E2 -7215.456} C_VEL
LIN {X 0,Y 474.662,Z 195.354,A -85,B 0,C 180,E1 -7219.01,E2 -7219.01} C_VEL
LIN {X 0,Y 474.591,Z 195.37,A -85,B 0,C 180,E1 -7221.729,E2 -7221.729} C_VEL
LIN {X 0,Y 474.629,Z 195.359,A -85,B 0,C 180,E1 -7224.495,E2 -7224.495} C_VEL
LIN {X 0,Y 474.603,Z 195.365,A -85,B 0,C 180,E1 -7227.326,E2 -7227.326} C_VEL
LIN {X 0,Y 474.6,Z 195.364,A -85,B 0,C 180,E1 -7230.231,E2 -7230.231} C_VEL
LIN {X 0,Y 474.617,Z 195.364,A -85,B 0,C 180,E1 -7233.222,E2 -7233.222} C_VEL
LIN {X 0,Y 474.586,Z 195.364,A -85,B 0,C 180,E1 -7236.324,E2 -7236.324} C_VEL
LIN {X 0,Y 474.625,Z 195.366,A -85,B 0,C 180,E1 -7239.548,E2 -7239.548} C_VEL
LIN {X 0,Y 474.579,Z 195.365,A -85,B 0,C 180,E1 -7242.23,E2 -7242.23} C_VEL
LIN {X 0,Y 474.618,Z 195.368,A -85,B 0,C 180,E1 -7245.298,E2 -7245.298} C_VEL
LIN {X 0,Y 474.594,Z 195.363,A -85,B 0,C 180,E1 -7248.211,E2 -7248.211} C_VEL
LIN {X 0,Y 474.61,Z 195.364,A -85,B 0,C 180,E1 -7251.542,E2 -7251.542} C_VEL
LIN {X 0,Y 474.622,Z 195.363,A -85,B 0,C 180,E1 -7254.725,E2 -7254.725} C_VEL
LIN {X 0,Y 474.628,Z 195.361,A -85,B 0,C 180,E1 -7257.787,E2 -7257.787} C_VEL
LIN {X 0,Y 474.601,Z 195.37,A -85,B 0,C 180,E1 -7260.89,E2 -7260.89} C_VEL
LIN {X 0,Y 474.651,Z 195.466,A -85,B 0,C 180,E1 -7262.445,E2 -7262.445} C_VEL
LIN {X 0,Y 477.035,Z 206.976,A -85,B 0,C 180,E1 -7264.404,E2 -7264.404} C_VEL
LIN {X 0,Y 477.17,Z 211.831,A -85,B 0,C 180,E1 -7265.18,E2 -7265.18} C_VEL
LIN {X 0,Y 476.322,Z 233.122,A -85,B 0,C 180,E1 -7268.476,E2 -7268.476} C_VEL
LIN {X 0,Y 475.578,Z 254.227,A -85,B 0,C 180,E1 -7271.698,E2 -7271.698} C_VEL
LIN {X 0,Y 475.248,Z 264.415,A -85,B 0,C 180,E1 -7273.241,E2 -7273.241} C_VEL
LIN {X 0,Y 477.88,Z 285.804,A -85,B 0,C 180,E1 -7273.683,E2 -7273.683} C_VEL
LIN {X 0,Y 477.159,Z 374.257,A -85,B 0,C 180,E1 -7275.09,E2 -7275.09} C_VEL
LIN {X 0,Y 476.752,Z 387.211,A -85,B 0,C 180,E1 -7275.459,E2 -7275.459} C_VEL
LIN {X 0,Y 476.337,Z 400.375,A -85,B 0,C 180,E1 -7276.019,E2 -7276.019} C_VEL
LIN {X 0,Y 475.768,Z 413.077,A -85,B 0,C 180,E1 -7276.764,E2 -7276.764} C_VEL
LIN {X 0,Y 475.266,Z 424.875,A -85,B 0,C 180,E1 -7277.657,E2 -7277.657} C_VEL
LIN {X 0,Y 474.905,Z 435.619,A -85,B 0,C 180,E1 -7278.692,E2 -7278.692} C_VEL
LIN {X 0,Y 474.45,Z 444.666,A -85,B 0,C 180,E1 -7279.761,E2 -7279.761} C_VEL
LIN {X 0,Y 474.184,Z 453.519,A -85,B 0,C 180,E1 -7281.047,E2 -7281.047} C_VEL
LIN {X 0,Y 473.996,Z 460.576,A -85,B 0,C 180,E1 -7282.331,E2 -7282.331} C_VEL
LIN {X 0,Y 473.9,Z 465.887,A -85,B 0,C 180,E1 -7283.526,E2 -7283.526} C_VEL
LIN {X 0,Y 473.834,Z 470.656,A -85,B 0,C 180,E1 -7284.894,E2 -7284.894} C_VEL
LIN {X 0,Y 473.792,Z 472.991,A -85,B 0,C 180,E1 -7285.746,E2 -7285.746} C_VEL
LIN {X 0,Y 473.861,Z 474.896,A -85,B 0,C 180,E1 -7286.599,E2 -7286.599} C_VEL
LIN {X 0,Y 473.877,Z 476.321,A -85,B 0,C 180,E1 -7287.45,E2 -7287.45} C_VEL
LIN {X 0,Y 473.723,Z 477.923,A -85,B 0,C 180,E1 -7289.15,E2 -7289.15} C_VEL
LIN {X 0,Y 473.725,Z 478.13,A -85,B 0,C 180,E1 -7290,E2 -7290} C_VEL
LIN {X 0,Y 473.724,Z 477.892,A -85,B 0,C 180,E1 -7290.85,E2 -7290.85} C_VEL
LIN {X 0,Y 473.879,Z 476.222,A -85,B 0,C 180,E1 -7292.55,E2 -7292.55} C_VEL
LIN {X 0,Y 473.876,Z 474.77,A -85,B 0,C 180,E1 -7293.401,E2 -7293.401} C_VEL
LIN {X 0,Y 473.783,Z 471.723,A -85,B 0,C 180,E1 -7294.68,E2 -7294.68} C_VEL
LIN {X 0,Y 473.831,Z 467.621,A -85,B 0,C 180,E1 -7295.959,E2 -7295.959} C_VEL
LIN {X 0,Y 473.998,Z 461.321,A -85,B 0,C 180,E1 -7297.454,E2 -7297.454} C_VEL
LIN {X 0,Y 474.122,Z 454.445,A -85,B 0,C 180,E1 -7298.739,E2 -7298.739} C_VEL
LIN {X 0,Y 474.387,Z 445.934,A -85,B 0,C 180,E1 -7300.025,E2 -7300.025} C_VEL
LIN {X 0,Y 474.795,Z 437.193,A -85,B 0,C 180,E1 -7301.094,E2 -7301.094} C_VEL
LIN {X 0,Y 475.155,Z 427.192,A -85,B 0,C 180,E1 -7302.098,E2 -7302.098} C_VEL
LIN {X 0,Y 475.648,Z 415.771,A -85,B 0,C 180,E1 -7303.022,E2 -7303.022} C_VEL
LIN {X 0,Y 476.106,Z 403.997,A -85,B 0,C 180,E1 -7303.77,E2 -7303.77} C_VEL
LIN {X 0,Y 476.557,Z 391.809,A -85,B 0,C 180,E1 -7304.356,E2 -7304.356} C_VEL
LIN {X 0,Y 477.003,Z 379.539,A -85,B 0,C 180,E1 -7304.778,E2 -7304.778} C_VEL
LIN {X 0,Y 477.276,Z 366.04,A -85,B 0,C 180,E1 -7305.069,E2 -7305.069} C_VEL
LIN {X 0,Y 477.751,Z 283.351,A -85,B 0,C 180,E1 -7306.38,E2 -7306.38} C_VEL
LIN {X 0,Y 475.144,Z 262.903,A -85,B 0,C 180,E1 -7306.821,E2 -7306.821} C_VEL
LIN {X 0,Y 475.768,Z 242.341,A -85,B 0,C 180,E1 -7309.862,E2 -7309.862} C_VEL
LIN {X 0,Y 476.293,Z 222.73,A -85,B 0,C 180,E1 -7312.789,E2 -7312.789} C_VEL
LIN {X 0,Y 476.81,Z 207.581,A -85,B 0,C 180,E1 -7315.072,E2 -7315.072} C_VEL
LIN {X 0,Y 475.564,Z 199.872,A -85,B 0,C 180,E1 -7316.317,E2 -7316.317} C_VEL
LIN {X 0,Y 474.652,Z 195.365,A -85,B 0,C 180,E1 -7317.084,E2 -7317.084} C_VEL
LIN {X 0,Y 474.595,Z 195.369,A -85,B 0,C 180,E1 -7320.231,E2 -7320.231} C_VEL
LIN {X 0,Y 474.625,Z 195.366,A -85,B 0,C 180,E1 -7323.221,E2 -7323.221} C_VEL
LIN {X 0,Y 474.584,Z 195.367,A -85,B 0,C 180,E1 -7326.324,E2 -7326.324} C_VEL
LIN {X 0,Y 474.622,Z 195.361,A -85,B 0,C 180,E1 -7329.548,E2 -7329.548} C_VEL
LIN {X 0,Y 474.598,Z 195.366,A -85,B 0,C 180,E1 -7332.233,E2 -7332.233} C_VEL
LIN {X 0,Y 474.616,Z 195.361,A -85,B 0,C 180,E1 -7335.298,E2 -7335.298} C_VEL
LIN {X 0,Y 474.609,Z 195.364,A -85,B 0,C 180,E1 -7338.213,E2 -7338.213} C_VEL
LIN {X 0,Y 474.608,Z 195.362,A -85,B 0,C 180,E1 -7341.542,E2 -7341.542} C_VEL
LIN {X 0,Y 474.622,Z 195.362,A -85,B 0,C 180,E1 -7344.725,E2 -7344.725} C_VEL
LIN {X 0,Y 474.635,Z 195.36,A -85,B 0,C 180,E1 -7347.788,E2 -7347.788} C_VEL
LIN {X 0,Y 474.607,Z 195.362,A -85,B 0,C 180,E1 -7350.888,E2 -7350.888} C_VEL
LIN {X 0,Y 474.613,Z 195.362,A -85,B 0,C 180,E1 -7353.625,E2 -7353.625} C_VEL
LIN {X 0,Y 474.634,Z 195.359,A -85,B 0,C 180,E1 -7356.642,E2 -7356.642} C_VEL
LIN {X 0,Y 474.653,Z 195.362,A -85,B 0,C 180,E1 -7360.089,E2 -7360.089} C_VEL
LIN {X 0,Y 474.633,Z 195.357,A -85,B 0,C 180,E1 -7362.774,E2 -7362.774} C_VEL
LIN {X 0,Y 474.642,Z 195.361,A -85,B 0,C 180,E1 -7365.421,E2 -7365.421} C_VEL
LIN {X 0,Y 474.705,Z 195.352,A -85,B 0,C 180,E1 -7368.037,E2 -7368.037} C_VEL
LIN {X 0,Y 474.727,Z 195.351,A -85,B 0,C 180,E1 -7371.486,E2 -7371.486} C_VEL
LIN {X 0,Y 474.771,Z 195.344,A -85,B 0,C 180,E1 -7374.052,E2 -7374.052} C_VEL
LIN {X 0,Y 474.894,Z 195.334,A -85,B 0,C 180,E1 -7377.455,E2 -7377.455} C_VEL
LIN {X 0,Y 474.912,Z 195.326,A -85,B 0,C 180,E1 -7380,E2 -7380} C_VEL
LIN {X 0,Y 474.894,Z 195.328,A -85,B 0,C 180,E1 -7382.545,E2 -7382.545} C_VEL
LIN {X 0,Y 474.762,Z 195.344,A -85,B 0,C 180,E1 -7385.948,E2 -7385.948} C_VEL
LIN {X 0,Y 474.711,Z 195.351,A -85,B 0,C 180,E1 -7388.514,E2 -7388.514} C_VEL
LIN {X 0,Y 474.705,Z 195.354,A -85,B 0,C 180,E1 -7391.962,E2 -7391.962} C_VEL
LIN {X 0,Y 474.7,Z 195.357,A -85,B 0,C 180,E1 -7395.456,E2 -7395.456} C_VEL
LIN {X 0,Y 474.666,Z 195.361,A -85,B 0,C 180,E1 -7399.01,E2 -7399.01} C_VEL
LIN {X 0,Y 474.706,Z 195.463,A -85,B 0,C 180,E1 -7400.615,E2 -7400.615} C_VEL
LIN {X 0,Y 475.434,Z 198.998,A -85,B 0,C 180,E1 -7401.268,E2 -7401.268} C_VEL
LIN {X 0,Y 478.185,Z 209.853,A -85,B 0,C 180,E1 -7401.557,E2 -7401.557} C_VEL
LIN {X 0,Y 478.185,Z 230.523,A -85,B 0,C 180,E1 -7401.898,E2 -7401.898} C_VEL
LIN {X 0,Y 477.467,Z 306.705,A -85,B 0,C 180,E1 -7403.13,E2 -7403.13} C_VEL
LIN {X 0,Y 477.263,Z 320.102,A -85,B 0,C 180,E1 -7403.528,E2 -7403.528} C_VEL
LIN {X 0,Y 476.96,Z 332.459,A -85,B 0,C 180,E1 -7404.068,E2 -7404.068} C_VEL
LIN {X 0,Y 476.62,Z 343.759,A -85,B 0,C 180,E1 -7404.734,E2 -7404.734} C_VEL
LIN {X 0,Y 476.122,Z 355.53,A -85,B 0,C 180,E1 -7405.622,E2 -7405.622} C_VEL
LIN {X 0,Y 475.747,Z 365.276,A -85,B 0,C 180,E1 -7406.543,E2 -7406.543} C_VEL
LIN {X 0,Y 475.334,Z 374.381,A -85,B 0,C 180,E1 -7407.6,E2 -7407.6} C_VEL
LIN {X 0,Y 474.958,Z 382.425,A -85,B 0,C 180,E1 -7408.745,E2 -7408.745} C_VEL
LIN {X 0,Y 474.657,Z 389.502,A -85,B 0,C 180,E1 -7409.981,E2 -7409.981} C_VEL
LIN {X 0,Y 474.416,Z 395.265,A -85,B 0,C 180,E1 -7411.231,E2 -7411.231} C_VEL
LIN {X 0,Y 474.147,Z 400.764,A -85,B 0,C 180,E1 -7412.77,E2 -7412.77} C_VEL
LIN {X 0,Y 473.979,Z 404.628,A -85,B 0,C 180,E1 -7414.295,E2 -7414.295} C_VEL
LIN {X 0,Y 473.878,Z 406.511,A -85,B 0,C 180,E1 -7415.344,E2 -7415.344} C_VEL
LIN {X 0,Y 473.791,Z 408.024,A -85,B 0,C 180,E1 -7416.773,E2 -7416.773} C_VEL
LIN {X 0,Y 473.768,Z 408.415,A -85,B 0,C 180,E1 -7418.167,E2 -7418.167} C_VEL
LIN {X 0,Y 473.791,Z 407.671,A -85,B 0,C 180,E1 -7419.631,E2 -7419.631} C_VEL
LIN {X 0,Y 473.85,Z 406.165,A -85,B 0,C 180,E1 -7420.851,E2 -7420.851} C_VEL
LIN {X 0,Y 474.041,Z 402.631,A -85,B 0,C 180,E1 -7422.539,E2 -7422.539} C_VEL
LIN {X 0,Y 474.15,Z 399.004,A -85,B 0,C 180,E1 -7423.754,E2 -7423.754} C_VEL
LIN {X 0,Y 474.359,Z 394.402,A -85,B 0,C 180,E1 -7424.959,E2 -7424.959} C_VEL
LIN {X 0,Y 474.536,Z 388.684,A -85,B 0,C 180,E1 -7426.164,E2 -7426.164} C_VEL
LIN {X 0,Y 474.893,Z 381.226,A -85,B 0,C 180,E1 -7427.435,E2 -7427.435} C_VEL
LIN {X 0,Y 475.317,Z 372.407,A -85,B 0,C 180,E1 -7428.642,E2 -7428.642} C_VEL
LIN {X 0,Y 475.742,Z 362.385,A -85,B 0,C 180,E1 -7429.749,E2 -7429.749} C_VEL
LIN {X 0,Y 476.144,Z 351.603,A -85,B 0,C 180,E1 -7430.71,E2 -7430.71} C_VEL
LIN {X 0,Y 476.598,Z 339.43,A -85,B 0,C 180,E1 -7431.555,E2 -7431.555} C_VEL
LIN {X 0,Y 476.892,Z 330.539,A -85,B 0,C 180,E1 -7432.047,E2 -7432.047} C_VEL
LIN {X 0,Y 476.336,Z 326.909,A -85,B 0,C 180,E1 -7432.24,E2 -7432.24} C_VEL
LIN {X 0,Y 470.988,Z 315.581,A -85,B 0,C 180,E1 -7432.858,E2 -7432.858} C_VEL
LIN {X 0,Y 470.415,Z 311.813,A -85,B 0,C 180,E1 -7432.992,E2 -7432.992} C_VEL
LIN {X 0,Y 470.581,Z 298.495,A -85,B 0,C 180,E1 -7433.284,E2 -7433.284} C_VEL
LIN {X 0,Y 471.367,Z 211.391,A -85,B 0,C 180,E1 -7434.675,E2 -7434.675} C_VEL
LIN {X 0,Y 468.77,Z 200.819,A -85,B 0,C 180,E1 -7434.943,E2 -7434.943} C_VEL
LIN {X 0,Y 467.977,Z 198.319,A -85,B 0,C 180,E1 -7435.039,E2 -7435.039} C_VEL
LIN {X 0,Y 467.621,Z 196.239,A -85,B 0,C 180,E1 -7435.503,E2 -7435.503} C_VEL
LIN {X 0,Y 467.568,Z 196.244,A -85,B 0,C 180,E1 -7438.955,E2 -7438.955} C_VEL
LIN {X 0,Y 467.629,Z 196.231,A -85,B 0,C 180,E1 -7442.463,E2 -7442.463} C_VEL
LIN {X 0,Y 467.569,Z 196.246,A -85,B 0,C 180,E1 -7445.111,E2 -7445.111} C_VEL
LIN {X 0,Y 467.534,Z 196.242,A -85,B 0,C 180,E1 -7447.926,E2 -7447.926} C_VEL
LIN {X 0,Y 467.622,Z 196.236,A -85,B 0,C 180,E1 -7450.692,E2 -7450.692} C_VEL
LIN {X 0,Y 467.639,Z 196.231,A -85,B 0,C 180,E1 -7454.305,E2 -7454.305} C_VEL
LIN {X 0,Y 467.657,Z 196.227,A -85,B 0,C 180,E1 -7457.855,E2 -7457.855} C_VEL
LIN {X 0,Y 467.67,Z 196.226,A -85,B 0,C 180,E1 -7461.357,E2 -7461.357} C_VEL
LIN {X 0,Y 467.724,Z 196.219,A -85,B 0,C 180,E1 -7463.963,E2 -7463.963} C_VEL
LIN {X 0,Y 467.853,Z 196.203,A -85,B 0,C 180,E1 -7467.417,E2 -7467.417} C_VEL
LIN {X 0,Y 467.882,Z 196.201,A -85,B 0,C 180,E1 -7470,E2 -7470} C_VEL
LIN {X 0,Y 467.849,Z 196.209,A -85,B 0,C 180,E1 -7472.583,E2 -7472.583} C_VEL
LIN {X 0,Y 467.722,Z 196.223,A -85,B 0,C 180,E1 -7476.038,E2 -7476.038} C_VEL
LIN {X 0,Y 467.672,Z 196.229,A -85,B 0,C 180,E1 -7478.643,E2 -7478.643} C_VEL
LIN {X 0,Y 467.658,Z 196.234,A -85,B 0,C 180,E1 -7482.146,E2 -7482.146} C_VEL
LIN {X 0,Y 467.64,Z 196.232,A -85,B 0,C 180,E1 -7485.695,E2 -7485.695} C_VEL
LIN {X 0,Y 467.623,Z 196.232,A -85,B 0,C 180,E1 -7489.308,E2 -7489.308} C_VEL
LIN {X 0,Y 467.536,Z 196.249,A -85,B 0,C 180,E1 -7492.074,E2 -7492.074} C_VEL
LIN {X 0,Y 467.57,Z 196.238,A -85,B 0,C 180,E1 -7494.89,E2 -7494.89} C_VEL
LIN {X 0,Y 467.582,Z 196.244,A -85,B 0,C 180,E1 -7497.772,E2 -7497.772} C_VEL
LIN {X 0,Y 467.569,Z 196.239,A -85,B 0,C 180,E1 -7501.045,E2 -7501.045} C_VEL
LIN {X 0,Y 467.59,Z 196.237,A -85,B 0,C 180,E1 -7504.242,E2 -7504.242} C_VEL
LIN {X 0,Y 467.545,Z 196.244,A -85,B 0,C 180,E1 -7507.186,E2 -7507.186} C_VEL
LIN {X 0,Y 467.561,Z 196.24,A -85,B 0,C 180,E1 -7510.267,E2 -7510.267} C_VEL
LIN {X 0,Y 467.562,Z 196.239,A -85,B 0,C 180,E1 -7512.564,E2 -7512.564} C_VEL
LIN {X 0,Y 467.567,Z 196.241,A -85,B 0,C 180,E1 -7515.053,E2 -7515.053} C_VEL
LIN {X 0,Y 467.569,Z 196.239,A -85,B 0,C 180,E1 -7518.596,E2 -7518.596} C_VEL
LIN {X 0,Y 467.565,Z 196.239,A -85,B 0,C 180,E1 -7521.955,E2 -7521.955} C_VEL
LIN {X 0,Y 467.56,Z 196.247,A -85,B 0,C 180,E1 -7525.167,E2 -7525.167} C_VEL
LIN {X 0,Y 467.584,Z 196.236,A -85,B 0,C 180,E1 -7528.26,E2 -7528.26} C_VEL
LIN {X 0,Y 467.55,Z 196.246,A -85,B 0,C 180,E1 -7531.249,E2 -7531.249} C_VEL
LIN {X 0,Y 467.595,Z 196.236,A -85,B 0,C 180,E1 -7534.397,E2 -7534.397} C_VEL
LIN {X 0,Y 467.578,Z 196.244,A -85,B 0,C 180,E1 -7536.996,E2 -7536.996} C_VEL
LIN {X 0,Y 467.624,Z 196.231,A -85,B 0,C 180,E1 -7539.777,E2 -7539.777} C_VEL
LIN {X 0,Y 467.596,Z 196.239,A -85,B 0,C 180,E1 -7542.506,E2 -7542.506} C_VEL
LIN {X 0,Y 467.6,Z 196.236,A -85,B 0,C 180,E1 -7545.196,E2 -7545.196} C_VEL
LIN {X 0,Y 467.66,Z 196.227,A -85,B 0,C 180,E1 -7547.855,E2 -7547.855} C_VEL
LIN {X 0,Y 467.67,Z 196.226,A -85,B 0,C 180,E1 -7551.357,E2 -7551.357} C_VEL
LIN {X 0,Y 467.715,Z 196.222,A -85,B 0,C 180,E1 -7553.962,E2 -7553.962} C_VEL
LIN {X 0,Y 467.852,Z 196.203,A -85,B 0,C 180,E1 -7557.417,E2 -7557.417} C_VEL
